gfCNCPoint2[10858] = {X 102.8887, Y 52.2397, Z -3.0000, A 0.000, B 0.000, C 0.000 }
gfCNCPoint2[10859] = {X 101.6641, Y 52.2655, Z -3.0000, A 0.000, B 0.000, C 0.000 }
gfCNCPoint2[10860] = {X 100.4526, Y 52.0855, Z -3.0000, A 0.000, B 0.000, C 0.000 }
gfCNCPoint2[10861] = {X 99.2883, Y 51.7050, Z -3.0000, A 0.000, B 0.000, C 0.000 }
gfCNCPoint2[10862] = {X 98.2043, Y 51.1347, Z -3.0000, A 0.000, B 0.000, C 0.000 }
gfCNCPoint2[10863] = {X 97.2313, Y 50.3907, Z -3.0000, A 0.000, B 0.000, C 0.000 }
gfCNCPoint2[10864] = {X 96.3865, Y 51.0508, Z -3.0000, A 0.000, B 0.000, C 0.000 }
gfCNCPoint2[10865] = {X 95.4539, Y 51.5797, Z -3.0000, A 0.000, B 0.000, C 0.000 }
gfCNCPoint2[10866] = {X 94.4538, Y 51.9659, Z -3.0000, A 0.000, B 0.000, C 0.000 }
gfCNCPoint2[10867] = {X 93.4078, Y 52.2011, Z -3.0000, A 0.000, B 0.000, C 0.000 }
gfCNCPoint2[10868] = {X 92.3385, Y 52.2800, Z -3.0000, A 0.000, B 0.000, C 0.000 }
gfCNCPoint2[10869] = {X 85.8951, Y 52.2800, Z -3.0000, A 0.000, B 0.000, C 0.000 }
gfCNCPoint2[10870] = {X 84.6852, Y 52.1788, Z -3.0000, A 0.000, B 0.000, C 0.000 }
gfCNCPoint2[10871] = {X 83.5090, Y 51.8779, Z -3.0000, A 0.000, B 0.000, C 0.000 }
gfCNCPoint2[10872] = {X 82.3992, Y 51.3857, Z -3.0000, A 0.000, B 0.000, C 0.000 }
gfCNCPoint2[10873] = {X 81.3866, Y 50.7159, Z -3.0000, A 0.000, B 0.000, C 0.000 }
gfCNCPoint2[10874] = {X 80.5223, Y 52.0937, Z -3.0000, A 0.000, B 0.000, C 0.000 }
gfCNCPoint2[10875] = {X 79.4808, Y 53.3429, Z -3.0000, A 0.000, B 0.000, C 0.000 }
gfCNCPoint2[10876] = {X 78.2809, Y 54.4408, Z -3.0000, A 0.000, B 0.000, C 0.000 }
gfCNCPoint2[10877] = {X 76.9444, Y 55.3676, Z -3.0000, A 0.000, B 0.000, C 0.000 }
gfCNCPoint2[10878] = {X 75.4955, Y 56.1065, Z -3.0000, A 0.000, B 0.000, C 0.000 }
gfCNCPoint2[10879] = {X 73.9605, Y 56.6440, Z -3.0000, A 0.000, B 0.000, C 0.000 }
gfCNCPoint2[10880] = {X 72.3672, Y 56.9705, Z -3.0000, A 0.000, B 0.000, C 0.000 }
gfCNCPoint2[10881] = {X 70.7445, Y 57.0800, Z -3.0000, A 0.000, B 0.000, C 0.000 }
gfCNCPoint2[10882] = {X 64.1851, Y 57.0800, Z -3.0000, A 0.000, B 0.000, C 0.000 }
gfCNCPoint2[10883] = {X 62.6628, Y 56.9837, Z -3.0000, A 0.000, B 0.000, C 0.000 }
gfCNCPoint2[10884] = {X 61.1646, Y 56.6963, Z -3.0000, A 0.000, B 0.000, C 0.000 }
gfCNCPoint2[10885] = {X 59.7147, Y 56.2224, Z -3.0000, A 0.000, B 0.000, C 0.000 }
gfCNCPoint2[10886] = {X 58.3360, Y 55.5695, Z -3.0000, A 0.000, B 0.000, C 0.000 }
gfCNCPoint2[10887] = {X 57.0507, Y 54.7481, Z -3.0000, A 0.000, B 0.000, C 0.000 }
gfCNCPoint2[10888] = {X 55.8790, Y 53.7713, Z -3.0000, A 0.000, B 0.000, C 0.000 }
gfCNCPoint2[10889] = {X 54.7074, Y 54.7481, Z -3.0000, A 0.000, B 0.000, C 0.000 }
gfCNCPoint2[10890] = {X 53.4220, Y 55.5695, Z -3.0000, A 0.000, B 0.000, C 0.000 }
gfCNCPoint2[10891] = {X 52.0434, Y 56.2224, Z -3.0000, A 0.000, B 0.000, C 0.000 }
gfCNCPoint2[10892] = {X 50.5934, Y 56.6963, Z -3.0000, A 0.000, B 0.000, C 0.000 }
gfCNCPoint2[10893] = {X 49.0953, Y 56.9837, Z -3.0000, A 0.000, B 0.000, C 0.000 }
gfCNCPoint2[10894] = {X 47.5729, Y 57.0800, Z -3.0000, A 0.000, B 0.000, C 0.000 }
gfCNCPoint2[10895] = {X 40.6393, Y 57.0800, Z -3.0000, A 0.000, B 0.000, C 0.000 }
gfCNCPoint2[10896] = {X 39.3237, Y 57.0081, Z -3.0000, A 0.000, B 0.000, C 0.000 }
gfCNCPoint2[10897] = {X 38.0238, Y 56.7934, Z -3.0000, A 0.000, B 0.000, C 0.000 }
gfCNCPoint2[10898] = {X 36.7550, Y 56.4385, Z -3.0000, A 0.000, B 0.000, C 0.000 }
gfCNCPoint2[10899] = {X 35.5323, Y 55.9474, Z -3.0000, A 0.000, B 0.000, C 0.000 }
gfCNCPoint2[10900] = {X 34.1223, Y 56.7816, Z -3.0000, A 0.000, B 0.000, C 0.000 }
gfCNCPoint2[10901] = {X 32.6361, Y 57.4711, Z -3.0000, A 0.000, B 0.000, C 0.000 }
gfCNCPoint2[10902] = {X 31.0886, Y 58.0091, Z -3.0000, A 0.000, B 0.000, C 0.000 }
gfCNCPoint2[10903] = {X 29.4952, Y 58.3901, Z -3.0000, A 0.000, B 0.000, C 0.000 }
gfCNCPoint2[10904] = {X 27.8718, Y 58.6104, Z -3.0000, A 0.000, B 0.000, C 0.000 }
gfCNCPoint2[10905] = {X 26.1298, Y 59.3568, Z -3.0000, A 0.000, B 0.000, C 0.000 }
gfCNCPoint2[10906] = {X 24.3546, Y 60.0200, Z -3.0000, A 0.000, B 0.000, C 0.000 }
gfCNCPoint2[10907] = {X 21.9380, Y 60.7953, Z -3.0000, A 0.000, B 0.000, C 0.000 }
gfCNCPoint2[10908] = {X 19.4715, Y 61.3930, Z -3.0000, A 0.000, B 0.000, C 0.000 }
gfCNCPoint2[10909] = {X 16.9680, Y 61.8098, Z -3.0000, A 0.000, B 0.000, C 0.000 }
gfCNCPoint2[10910] = {X 14.4409, Y 62.0436, Z -3.0000, A 0.000, B 0.000, C 0.000 }
gfCNCPoint2[10911] = {X 11.9035, Y 62.0931, Z -3.0000, A 0.000, B 0.000, C 0.000 }
gfCNCPoint2[10912] = {X 11.9035, Y 88.0950, Z -3.0000, A 0.000, B 0.000, C 0.000 }
gfCNCPoint2[10913] = {X 113.6337, Y 88.0950, Z -3.0000, A 0.000, B 0.000, C 0.000 }
gfCNCPoint2[10914] = {X 114.7670, Y 86.8212, Z -3.0000, A 0.000, B 0.000, C 0.000 }
gfCNCPoint2[10915] = {X 116.0421, Y 85.6894, Z -3.0000, A 0.000, B 0.000, C 0.000 }
gfCNCPoint2[10916] = {X 117.4414, Y 84.7153, Z -3.0000, A 0.000, B 0.000, C 0.000 }
gfCNCPoint2[10917] = {X 118.9454, Y 83.9125, Z -3.0000, A 0.000, B 0.000, C 0.000 }
gfCNCPoint2[10918] = {X 120.5335, Y 83.2920, Z -3.0000, A 0.000, B 0.000, C 0.000 }
gfCNCPoint2[10919] = {X 122.1834, Y 82.8625, Z -3.0000, A 0.000, B 0.000, C 0.000 }
gfCNCPoint2[10920] = {X 144.8180, Y 58.0066, Z -3.0000, A 0.000, B 0.000, C 0.000 }
gfCNCPoint2[10921] = {X 144.9143, Y 56.3321, Z -3.0000, A 0.000, B 0.000, C 0.000 }
gfCNCPoint2[10922] = {X 145.2037, Y 54.6800, Z -3.0000, A 0.000, B 0.000, C 0.000 }
gfCNCPoint2[10923] = {X 143.0396, Y 54.6800, Z -3.0000, A 0.000, B 0.000, C 0.000 }
gfCNCPoint2[10924] = {X 142.7952, Y 54.6769, Z -3.0000, A 0.000, B 0.000, C 0.000 }
gfCNCPoint2[10925] = {X 142.5510, Y 54.6677, Z -3.0000, A 0.000, B 0.000, C 0.000 }
gfCNCPoint2[10926] = {X 141.0979, Y 54.4832, Z -3.0000, A 0.000, B 0.000, C 0.000 }
gfCNCPoint2[10927] = {X 139.6893, Y 54.0817, Z -3.0000, A 0.000, B 0.000, C 0.000 }
gfCNCPoint2[10928] = {X 138.3574, Y 53.4722, Z -3.0000, A 0.000, B 0.000, C 0.000 }
gfCNCPoint2[10929] = {X 137.1327, Y 52.6688, Z -3.0000, A 0.000, B 0.000, C 0.000 }
gfCNCPoint2[10930] = {X 136.0432, Y 51.6898, Z -3.0000, A 0.000, B 0.000, C 0.000 }
gfCNCPoint2[10931] = {X 135.1140, Y 50.5575, Z -3.0000, A 0.000, B 0.000, C 0.000 }
gfCNCPoint2[10932] = {X 134.3662, Y 49.2981, Z -3.0000, A 0.000, B 0.000, C 0.000 }
gfCNCPoint2[10933] = {X 133.8170, Y 47.9402, Z -3.0000, A 0.000, B 0.000, C 0.000 }
gfCNCPoint2[10934] = {X 133.4789, Y 46.5151, Z -3.0000, A 0.000, B 0.000, C 0.000 }
gfCNCPoint2[10935] = {X 133.3598, Y 45.0552, Z -3.0000, A 0.000, B 0.000, C 0.000 }
gfCNCPoint2[10936] = {X 133.3601, Y 44.1105, Z -3.0000, A 0.000, B 0.000, C 0.000 }
gfCNCPoint2[10937] = {X 133.4665, Y 42.7743, Z -3.0000, A 0.000, B 0.000, C 0.000 }
gfCNCPoint2[10938] = {X 133.7565, Y 41.4655, Z -3.0000, A 0.000, B 0.000, C 0.000 }
gfCNCPoint2[10939] = {X 136.0581, Y 42.1457, Z -3.0000, A 0.000, B 0.000, C 0.000 }
gfCNCPoint2[10940] = {X 136.3664, Y 41.2990, Z -3.0000, A 0.000, B 0.000, C 0.000 }
gfCNCPoint2[10941] = {X 136.7770, Y 40.4969, Z -3.0000, A 0.000, B 0.000, C 0.000 }
gfCNCPoint2[10942] = {X 137.2836, Y 39.7516, Z -3.0000, A 0.000, B 0.000, C 0.000 }
gfCNCPoint2[10943] = {X 137.2836, Y 23.8768, Z -3.0000, A 0.000, B 0.000, C 0.000 }
gfCNCPoint2[10944] = {X 136.4352, Y 24.2641, Z -3.0000, A 0.000, B 0.000, C 0.000 }
gfCNCPoint2[10945] = {X 135.5443, Y 24.5398, Z -3.0000, A 0.000, B 0.000, C 0.000 }
gfCNCPoint2[10946] = {X 134.6254, Y 24.6993, Z -3.0000, A 0.000, B 0.000, C 0.000 }
gfCNCPoint2[10947] = {X 134.2595, Y 24.7296, Z -3.0000, A 0.000, B 0.000, C 0.000 }
gfCNCPoint2[10948] = {X 133.8926, Y 24.7414, Z -3.0000, A 0.000, B 0.000, C 0.000 }
gfCNCPoint2[10949] = {X 133.2006, Y 24.7415, Z -3.0000, A 0.000, B 0.000, C 0.000 }
gfCNCPoint2[10950] = {X 131.9926, Y 24.6406, Z -3.0000, A 0.000, B 0.000, C 0.000 }
gfCNCPoint2[10951] = {X 130.8180, Y 24.3406, Z -3.0000, A 0.000, B 0.000, C 0.000 }
gfCNCPoint2[10952] = {X 129.7095, Y 23.8498, Z -3.0000, A 0.000, B 0.000, C 0.000 }
gfCNCPoint2[10953] = {X 128.6978, Y 23.1819, Z -3.0000, A 0.000, B 0.000, C 0.000 }
gfCNCPoint2[10954] = {X 127.8110, Y 22.3554, Z -3.0000, A 0.000, B 0.000, C 0.000 }
gfCNCPoint2[10955] = {X 127.0736, Y 21.3931, Z -3.0000, A 0.000, B 0.000, C 0.000 }
gfCNCPoint2[10956] = {X 126.5061, Y 20.3219, Z -3.0000, A 0.000, B 0.000, C 0.000 }
gfCNCPoint2[10957] = {X 126.1243, Y 19.1713, Z -3.0000, A 0.000, B 0.000, C 0.000 }
gfCNCPoint2[10958] = {X 125.9387, Y 17.9733, Z -3.0000, A 0.000, B 0.000, C 0.000 }
gfCNCPoint2[10959] = {X 125.9251, Y 17.7176, Z -3.0000, A 0.000, B 0.000, C 0.000 }
gfCNCPoint2[10960] = {X 125.9206, Y 17.4615, Z -3.0000, A 0.000, B 0.000, C 0.000 }
gfCNCPoint2[10961] = {X 125.9206, Y 10.4835, Z -3.0000, A 0.000, B 0.000, C 0.000 }
gfCNCPoint2[10962] = {X 125.9372, Y 9.9932, Z -3.0000, A 0.000, B 0.000, C 0.000 }
gfCNCPoint2[10963] = {X 125.9867, Y 9.5050, Z -3.0000, A 0.000, B 0.000, C 0.000 }
gfCNCPoint2[10964] = {X 121.8686, Y 9.5050, Z -3.0000, A 0.000, B 0.000, C 0.000 }
gfCNCPoint2[10965] = {X 122.3091, Y 10.3411, Z -3.0000, A 0.000, B 0.000, C 0.000 }
gfCNCPoint2[10966] = {X 122.5801, Y 11.2463, Z -3.0000, A 0.000, B 0.000, C 0.000 }
gfCNCPoint2[10967] = {X 122.6716, Y 12.1868, Z -3.0000, A 0.000, B 0.000, C 0.000 }
gfCNCPoint2[10968] = {X 122.6714, Y 13.0237, Z -3.0000, A 0.000, B 0.000, C 0.000 }
gfCNCPoint2[10969] = {X 122.5640, Y 13.9970, Z -3.0000, A 0.000, B 0.000, C 0.000 }
gfCNCPoint2[10970] = {X 122.2645, Y 14.9292, Z -3.0000, A 0.000, B 0.000, C 0.000 }
gfCNCPoint2[10971] = {X 121.7850, Y 15.7828, Z -3.0000, A 0.000, B 0.000, C 0.000 }
gfCNCPoint2[10972] = {X 121.1447, Y 16.5236, Z -3.0000, A 0.000, B 0.000, C 0.000 }
gfCNCPoint2[10973] = {X 121.1435, Y 40.6621, Z -3.0000, A 0.000, B 0.000, C 0.000 }
gfCNCPoint2[10974] = {X 121.7851, Y 41.4041, Z -3.0000, A 0.000, B 0.000, C 0.000 }
gfCNCPoint2[10975] = {X 122.2653, Y 42.2595, Z -3.0000, A 0.000, B 0.000, C 0.000 }
gfCNCPoint2[10976] = {X 122.5648, Y 43.1936, Z -3.0000, A 0.000, B 0.000, C 0.000 }
gfCNCPoint2[10977] = {X 122.6714, Y 44.1688, Z -3.0000, A 0.000, B 0.000, C 0.000 }
gfCNCPoint2[10978] = {X 122.6716, Y 45.0000, Z -3.0000, A 0.000, B 0.000, C 0.000 }
gfCNCPoint2[10979] = {X 122.5778, Y 45.9520, Z -3.0000, A 0.000, B 0.000, C 0.000 }
gfCNCPoint2[10980] = {X 122.3001, Y 46.8675, Z -3.0000, A 0.000, B 0.000, C 0.000 }
gfCNCPoint2[10981] = {X 121.8491, Y 47.7112, Z -3.0000, A 0.000, B 0.000, C 0.000 }
gfCNCPoint2[10982] = {X 121.2423, Y 48.4507, Z -3.0000, A 0.000, B 0.000, C 0.000 }
gfCNCPoint2[10983] = {X 120.5028, Y 49.0576, Z -3.0000, A 0.000, B 0.000, C 0.000 }
gfCNCPoint2[10984] = {X 119.6591, Y 49.5085, Z -3.0000, A 0.000, B 0.000, C 0.000 }
gfCNCPoint2[10985] = {X 118.7436, Y 49.7862, Z -3.0000, A 0.000, B 0.000, C 0.000 }
gfCNCPoint2[10986] = {X 117.7916, Y 49.8800, Z -3.0000, A 0.000, B 0.000, C 0.000 }
gfCNCPoint2[10987] = {X 111.9185, Y 49.8800, Z -3.0000, A 0.000, B 0.000, C 0.000 }
gfCNCPoint2[10988] = {X 111.0234, Y 49.7972, Z -3.0000, A 0.000, B 0.000, C 0.000 }
gfCNCPoint2[10989] = {X 110.1587, Y 49.5517, Z -3.0000, A 0.000, B 0.000, C 0.000 }
gfCNCPoint2[10990] = {X 109.3537, Y 49.1517, Z -3.0000, A 0.000, B 0.000, C 0.000 }
gfCNCPoint2[10991] = {X 108.6357, Y 48.6108, Z -3.0000, A 0.000, B 0.000, C 0.000 }
gfCNCPoint2[10992] = {X 108.0714, Y 48.0024, Z -3.0000, A 0.000, B 0.000, C 0.000 }
gfCNCPoint2[10993] = {X 107.6183, Y 47.3071, Z -3.0000, A 0.000, B 0.000, C 0.000 }
gfCNCPoint2[10994] = {X 107.2895, Y 46.5451, Z -3.0000, A 0.000, B 0.000, C 0.000 }
gfCNCPoint2[10995] = {X 107.0947, Y 45.7384, Z -3.0000, A 0.000, B 0.000, C 0.000 }
gfCNCPoint2[10996] = {X 106.6287, Y 46.8769, Z -3.0000, A 0.000, B 0.000, C 0.000 }
gfCNCPoint2[10997] = {X 106.1131, Y 47.8110, Z -3.0000, A 0.000, B 0.000, C 0.000 }
gfCNCPoint2[10998] = {X 105.4068, Y 48.6108, Z -3.0000, A 0.000, B 0.000, C 0.000 }
gfCNCPoint2[10999] = {X 104.8391, Y 49.0550, Z -3.0000, A 0.000, B 0.000, C 0.000 }
gfCNCPoint2[11000] = {X 104.2121, Y 49.4107, Z -3.0000, A 0.000, B 0.000, C 0.000 }
gfCNCPoint2[11001] = {X 103.3106, Y 49.7335, Z -3.0000, A 0.000, B 0.000, C 0.000 }
gfCNCPoint2[11002] = {X 102.3635, Y 49.8741, Z -3.0000, A 0.000, B 0.000, C 0.000 }
gfCNCPoint2[11003] = {X 101.4071, Y 49.8271, Z -3.0000, A 0.000, B 0.000, C 0.000 }
gfCNCPoint2[11004] = {X 100.4784, Y 49.5941, Z -3.0000, A 0.000, B 0.000, C 0.000 }
gfCNCPoint2[11005] = {X 99.6130, Y 49.1844, Z -3.0000, A 0.000, B 0.000, C 0.000 }
gfCNCPoint2[11006] = {X 98.8443, Y 48.6135, Z -3.0000, A 0.000, B 0.000, C 0.000 }
gfCNCPoint2[11007] = {X 98.1362, Y 47.8127, Z -3.0000, A 0.000, B 0.000, C 0.000 }
gfCNCPoint2[11008] = {X 97.6194, Y 46.8769, Z -3.0000, A 0.000, B 0.000, C 0.000 }
gfCNCPoint2[11009] = {X 97.1600, Y 45.7536, Z -3.0000, A 0.000, B 0.000, C 0.000 }
gfCNCPoint2[11010] = {X 96.9635, Y 46.5570, Z -3.0000, A 0.000, B 0.000, C 0.000 }
gfCNCPoint2[11011] = {X 96.6342, Y 47.3156, Z -3.0000, A 0.000, B 0.000, C 0.000 }
gfCNCPoint2[11012] = {X 96.1814, Y 48.0078, Z -3.0000, A 0.000, B 0.000, C 0.000 }
gfCNCPoint2[11013] = {X 95.6183, Y 48.6135, Z -3.0000, A 0.000, B 0.000, C 0.000 }
gfCNCPoint2[11014] = {X 94.9007, Y 49.1533, Z -3.0000, A 0.000, B 0.000, C 0.000 }
gfCNCPoint2[11015] = {X 94.0964, Y 49.5524, Z -3.0000, A 0.000, B 0.000, C 0.000 }
gfCNCPoint2[11016] = {X 93.2326, Y 49.7974, Z -3.0000, A 0.000, B 0.000, C 0.000 }
gfCNCPoint2[11017] = {X 92.3385, Y 49.8800, Z -3.0000, A 0.000, B 0.000, C 0.000 }
gfCNCPoint2[11018] = {X 85.8951, Y 49.8800, Z -3.0000, A 0.000, B 0.000, C 0.000 }
gfCNCPoint2[11019] = {X 85.0841, Y 49.8121, Z -3.0000, A 0.000, B 0.000, C 0.000 }
gfCNCPoint2[11020] = {X 84.2956, Y 49.6104, Z -3.0000, A 0.000, B 0.000, C 0.000 }
gfCNCPoint2[11021] = {X 83.5517, Y 49.2805, Z -3.0000, A 0.000, B 0.000, C 0.000 }
gfCNCPoint2[11022] = {X 82.8729, Y 48.8316, Z -3.0000, A 0.000, B 0.000, C 0.000 }
gfCNCPoint2[11023] = {X 82.2391, Y 48.2324, Z -3.0000, A 0.000, B 0.000, C 0.000 }
gfCNCPoint2[11024] = {X 81.7221, Y 47.5300, Z -3.0000, A 0.000, B 0.000, C 0.000 }
gfCNCPoint2[11025] = {X 81.3384, Y 46.7467, Z -3.0000, A 0.000, B 0.000, C 0.000 }
gfCNCPoint2[11026] = {X 81.1002, Y 45.9077, Z -3.0000, A 0.000, B 0.000, C 0.000 }
gfCNCPoint2[11027] = {X 81.0152, Y 45.0397, Z -3.0000, A 0.000, B 0.000, C 0.000 }
gfCNCPoint2[11028] = {X 81.0151, Y 44.2034, Z -3.0000, A 0.000, B 0.000, C 0.000 }
gfCNCPoint2[11029] = {X 81.1203, Y 43.2199, Z -3.0000, A 0.000, B 0.000, C 0.000 }
gfCNCPoint2[11030] = {X 81.4192, Y 42.2770, Z -3.0000, A 0.000, B 0.000, C 0.000 }
gfCNCPoint2[11031] = {X 81.9000, Y 41.4125, Z -3.0000, A 0.000, B 0.000, C 0.000 }
gfCNCPoint2[11032] = {X 82.5434, Y 40.6612, Z -3.0000, A 0.000, B 0.000, C 0.000 }
gfCNCPoint2[11033] = {X 82.5432, Y 25.2537, Z -3.0000, A 0.000, B 0.000, C 0.000 }
gfCNCPoint2[11034] = {X 77.7432, Y 25.2537, Z -3.0000, A 0.000, B 0.000, C 0.000 }
gfCNCPoint2[11035] = {X 77.7431, Y 18.1980, Z -3.0000, A 0.000, B 0.000, C 0.000 }
gfCNCPoint2[11036] = {X 77.0784, Y 16.9741, Z -3.0000, A 0.000, B 0.000, C 0.000 }
gfCNCPoint2[11037] = {X 76.5962, Y 15.6674, Z -3.0000, A 0.000, B 0.000, C 0.000 }
gfCNCPoint2[11038] = {X 76.3065, Y 14.3050, Z -3.0000, A 0.000, B 0.000, C 0.000 }
gfCNCPoint2[11039] = {X 74.0412, Y 14.3050, Z -3.0000, A 0.000, B 0.000, C 0.000 }
gfCNCPoint2[11040] = {X 73.9992, Y 14.7015, Z -3.0000, A 0.000, B 0.000, C 0.000 }
gfCNCPoint2[11041] = {X 73.9463, Y 15.0967, Z -3.0000, A 0.000, B 0.000, C 0.000 }
gfCNCPoint2[11042] = {X 77.7432, Y 25.2537, Z -3.0000, A 0.000, B 0.000, C 0.000 }
gfCNCPoint2[11043] = {X 80.1432, Y 25.2537, Z -3.0000, A 0.000, B 0.000, C 0.000 }
gfCNCPoint2[11044] = {X 80.1431, Y 17.4405, Z -3.0000, A 0.000, B 0.000, C 0.000 }
gfCNCPoint2[11045] = {X 79.4946, Y 16.4468, Z -3.0000, A 0.000, B 0.000, C 0.000 }
gfCNCPoint2[11046] = {X 79.0161, Y 15.3611, Z -3.0000, A 0.000, B 0.000, C 0.000 }
gfCNCPoint2[11047] = {X 78.7204, Y 14.2120, Z -3.0000, A 0.000, B 0.000, C 0.000 }
gfCNCPoint2[11048] = {X 78.6153, Y 13.0301, Z -3.0000, A 0.000, B 0.000, C 0.000 }
gfCNCPoint2[11049] = {X 78.6151, Y 12.1868, Z -3.0000, A 0.000, B 0.000, C 0.000 }
gfCNCPoint2[11050] = {X 78.6164, Y 12.0459, Z -3.0000, A 0.000, B 0.000, C 0.000 }
gfCNCPoint2[11051] = {X 78.6205, Y 11.9050, Z -3.0000, A 0.000, B 0.000, C 0.000 }
gfCNCPoint2[11052] = {X 71.6988, Y 11.9050, Z -3.0000, A 0.000, B 0.000, C 0.000 }
gfCNCPoint2[11053] = {X 71.7013, Y 12.0459, Z -3.0000, A 0.000, B 0.000, C 0.000 }
gfCNCPoint2[11054] = {X 71.7021, Y 12.1868, Z -3.0000, A 0.000, B 0.000, C 0.000 }
gfCNCPoint2[11055] = {X 71.7016, Y 13.0911, Z -3.0000, A 0.000, B 0.000, C 0.000 }
gfCNCPoint2[11056] = {X 71.6385, Y 14.2157, Z -3.0000, A 0.000, B 0.000, C 0.000 }
gfCNCPoint2[11057] = {X 71.4711, Y 15.3294, Z -3.0000, A 0.000, B 0.000, C 0.000 }
gfCNCPoint2[11058] = {X 78.9542, Y 35.3473, Z -3.0000, A 0.000, B 0.000, C 0.000 }
gfCNCPoint2[11059] = {X 79.5718, Y 35.9623, Z -3.0000, A 0.000, B 0.000, C 0.000 }
gfCNCPoint2[11060] = {X 80.1433, Y 36.6202, Z -3.0000, A 0.000, B 0.000, C 0.000 }
gfCNCPoint2[11061] = {X 80.1432, Y 25.2537, Z -3.0000, A 0.000, B 0.000, C 0.000 }
gfCNCPoint2[11062] = {X 82.5432, Y 25.2537, Z -3.0000, A 0.000, B 0.000, C 0.000 }
gfCNCPoint2[11063] = {X 82.5431, Y 16.5247, Z -3.0000, A 0.000, B 0.000, C 0.000 }
gfCNCPoint2[11064] = {X 81.9017, Y 15.7830, Z -3.0000, A 0.000, B 0.000, C 0.000 }
gfCNCPoint2[11065] = {X 81.4216, Y 14.9280, Z -3.0000, A 0.000, B 0.000, C 0.000 }
gfCNCPoint2[11066] = {X 81.1221, Y 13.9943, Z -3.0000, A 0.000, B 0.000, C 0.000 }
gfCNCPoint2[11067] = {X 81.0153, Y 13.0196, Z -3.0000, A 0.000, B 0.000, C 0.000 }
gfCNCPoint2[11068] = {X 81.0151, Y 12.1868, Z -3.0000, A 0.000, B 0.000, C 0.000 }
gfCNCPoint2[11069] = {X 81.0160, Y 12.0924, Z -3.0000, A 0.000, B 0.000, C 0.000 }
gfCNCPoint2[11070] = {X 81.0187, Y 11.9979, Z -3.0000, A 0.000, B 0.000, C 0.000 }
gfCNCPoint2[11071] = {X 81.1324, Y 11.1230, Z -3.0000, A 0.000, B 0.000, C 0.000 }
gfCNCPoint2[11072] = {X 81.4018, Y 10.2829, Z -3.0000, A 0.000, B 0.000, C 0.000 }
gfCNCPoint2[11073] = {X 81.8180, Y 9.5050, Z -3.0000, A 0.000, B 0.000, C 0.000 }
gfCNCPoint2[11074] = {X 82.2190, Y 9.7688, Z -3.0000, A 0.000, B 0.000, C 0.000 }
gfCNCPoint2[11075] = {X 82.7659, Y 9.0936, Z -3.0000, A 0.000, B 0.000, C 0.000 }
gfCNCPoint2[11076] = {X 83.4347, Y 8.5390, Z -3.0000, A 0.000, B 0.000, C 0.000 }
gfCNCPoint2[11077] = {X 84.1995, Y 8.1266, Z -3.0000, A 0.000, B 0.000, C 0.000 }
gfCNCPoint2[11078] = {X 85.0304, Y 7.8726, Z -3.0000, A 0.000, B 0.000, C 0.000 }
gfCNCPoint2[11079] = {X 85.8951, Y 7.7868, Z -3.0000, A 0.000, B 0.000, C 0.000 }
gfCNCPoint2[11080] = {X 94.0497, Y 7.7868, Z -3.0000, A 0.000, B 0.000, C 0.000 }
gfCNCPoint2[11081] = {X 95.0288, Y 7.8971, Z -3.0000, A 0.000, B 0.000, C 0.000 }
gfCNCPoint2[11082] = {X 95.9588, Y 8.2226, Z -3.0000, A 0.000, B 0.000, C 0.000 }
gfCNCPoint2[11083] = {X 96.7930, Y 8.7468, Z -3.0000, A 0.000, B 0.000, C 0.000 }
gfCNCPoint2[11084] = {X 97.4897, Y 9.4435, Z -3.0000, A 0.000, B 0.000, C 0.000 }
gfCNCPoint2[11085] = {X 98.0139, Y 10.2777, Z -3.0000, A 0.000, B 0.000, C 0.000 }
gfCNCPoint2[11086] = {X 98.3394, Y 11.2077, Z -3.0000, A 0.000, B 0.000, C 0.000 }
gfCNCPoint2[11087] = {X 98.4497, Y 12.1868, Z -3.0000, A 0.000, B 0.000, C 0.000 }
gfCNCPoint2[11088] = {X 98.4494, Y 13.0233, Z -3.0000, A 0.000, B 0.000, C 0.000 }
gfCNCPoint2[11089] = {X 98.3723, Y 13.7994, Z -3.0000, A 0.000, B 0.000, C 0.000 }
gfCNCPoint2[11090] = {X 98.1594, Y 14.5497, Z -3.0000, A 0.000, B 0.000, C 0.000 }
gfCNCPoint2[11091] = {X 97.8174, Y 15.2505, Z -3.0000, A 0.000, B 0.000, C 0.000 }
gfCNCPoint2[11092] = {X 98.3672, Y 16.6193, Z -3.0000, A 0.000, B 0.000, C 0.000 }
gfCNCPoint2[11093] = {X 101.8765, Y 25.3184, Z -3.0000, A 0.000, B 0.000, C 0.000 }
gfCNCPoint2[11094] = {X 105.9244, Y 15.2235, Z -3.0000, A 0.000, B 0.000, C 0.000 }
gfCNCPoint2[11095] = {X 105.5858, Y 14.5158, Z -3.0000, A 0.000, B 0.000, C 0.000 }
gfCNCPoint2[11096] = {X 105.3782, Y 13.7593, Z -3.0000, A 0.000, B 0.000, C 0.000 }
gfCNCPoint2[11097] = {X 105.3083, Y 12.9779, Z -3.0000, A 0.000, B 0.000, C 0.000 }
gfCNCPoint2[11098] = {X 105.3083, Y 12.1868, Z -3.0000, A 0.000, B 0.000, C 0.000 }
gfCNCPoint2[11099] = {X 105.4186, Y 11.2077, Z -3.0000, A 0.000, B 0.000, C 0.000 }
gfCNCPoint2[11100] = {X 105.7440, Y 10.2777, Z -3.0000, A 0.000, B 0.000, C 0.000 }
gfCNCPoint2[11101] = {X 106.2682, Y 9.4435, Z -3.0000, A 0.000, B 0.000, C 0.000 }
gfCNCPoint2[11102] = {X 106.9649, Y 8.7468, Z -3.0000, A 0.000, B 0.000, C 0.000 }
gfCNCPoint2[11103] = {X 107.7992, Y 8.2226, Z -3.0000, A 0.000, B 0.000, C 0.000 }
gfCNCPoint2[11104] = {X 108.7292, Y 7.8971, Z -3.0000, A 0.000, B 0.000, C 0.000 }
gfCNCPoint2[11105] = {X 109.7083, Y 7.7868, Z -3.0000, A 0.000, B 0.000, C 0.000 }
gfCNCPoint2[11106] = {X 117.7916, Y 7.7868, Z -3.0000, A 0.000, B 0.000, C 0.000 }
gfCNCPoint2[11107] = {X 118.7707, Y 7.8971, Z -3.0000, A 0.000, B 0.000, C 0.000 }
gfCNCPoint2[11108] = {X 119.7007, Y 8.2226, Z -3.0000, A 0.000, B 0.000, C 0.000 }
gfCNCPoint2[11109] = {X 120.5349, Y 8.7468, Z -3.0000, A 0.000, B 0.000, C 0.000 }
gfCNCPoint2[11110] = {X 121.2316, Y 9.4435, Z -3.0000, A 0.000, B 0.000, C 0.000 }
gfCNCPoint2[11111] = {X 121.7558, Y 10.2777, Z -3.0000, A 0.000, B 0.000, C 0.000 }
gfCNCPoint2[11112] = {X 122.0813, Y 11.2077, Z -3.0000, A 0.000, B 0.000, C 0.000 }
gfCNCPoint2[11113] = {X 122.1916, Y 12.1868, Z -3.0000, A 0.000, B 0.000, C 0.000 }
gfCNCPoint2[11114] = {X 122.1913, Y 13.0233, Z -3.0000, A 0.000, B 0.000, C 0.000 }
gfCNCPoint2[11115] = {X 122.0831, Y 13.9491, Z -3.0000, A 0.000, B 0.000, C 0.000 }
gfCNCPoint2[11116] = {X 121.7822, Y 14.8314, Z -3.0000, A 0.000, B 0.000, C 0.000 }
gfCNCPoint2[11117] = {X 121.3022, Y 15.6305, Z -3.0000, A 0.000, B 0.000, C 0.000 }
gfCNCPoint2[11118] = {X 120.6647, Y 16.3105, Z -3.0000, A 0.000, B 0.000, C 0.000 }
gfCNCPoint2[11119] = {X 120.6635, Y 40.8758, Z -3.0000, A 0.000, B 0.000, C 0.000 }
gfCNCPoint2[11120] = {X 120.6784, Y 40.8882, Z -3.0000, A 0.000, B 0.000, C 0.000 }
gfCNCPoint2[11121] = {X 121.3172, Y 41.5763, Z -3.0000, A 0.000, B 0.000, C 0.000 }
gfCNCPoint2[11122] = {X 121.7955, Y 42.3843, Z -3.0000, A 0.000, B 0.000, C 0.000 }
gfCNCPoint2[11123] = {X 122.0914, Y 43.2754, Z -3.0000, A 0.000, B 0.000, C 0.000 }
gfCNCPoint2[11124] = {X 122.1916, Y 44.2089, Z -3.0000, A 0.000, B 0.000, C 0.000 }
gfCNCPoint2[11125] = {X 122.1916, Y 45.0000, Z -3.0000, A 0.000, B 0.000, C 0.000 }
gfCNCPoint2[11126] = {X 122.0813, Y 45.9791, Z -3.0000, A 0.000, B 0.000, C 0.000 }
gfCNCPoint2[11127] = {X 121.7558, Y 46.9091, Z -3.0000, A 0.000, B 0.000, C 0.000 }
gfCNCPoint2[11128] = {X 121.2316, Y 47.7434, Z -3.0000, A 0.000, B 0.000, C 0.000 }
gfCNCPoint2[11129] = {X 120.5349, Y 48.4401, Z -3.0000, A 0.000, B 0.000, C 0.000 }
gfCNCPoint2[11130] = {X 119.7007, Y 48.9643, Z -3.0000, A 0.000, B 0.000, C 0.000 }
gfCNCPoint2[11131] = {X 118.7707, Y 49.2897, Z -3.0000, A 0.000, B 0.000, C 0.000 }
gfCNCPoint2[11132] = {X 117.7916, Y 49.4000, Z -3.0000, A 0.000, B 0.000, C 0.000 }
gfCNCPoint2[11133] = {X 111.9185, Y 49.4000, Z -3.0000, A 0.000, B 0.000, C 0.000 }
gfCNCPoint2[11134] = {X 110.9394, Y 49.2897, Z -3.0000, A 0.000, B 0.000, C 0.000 }
gfCNCPoint2[11135] = {X 110.0094, Y 48.9643, Z -3.0000, A 0.000, B 0.000, C 0.000 }
gfCNCPoint2[11136] = {X 109.1751, Y 48.4400, Z -3.0000, A 0.000, B 0.000, C 0.000 }
gfCNCPoint2[11137] = {X 108.4784, Y 47.7433, Z -3.0000, A 0.000, B 0.000, C 0.000 }
gfCNCPoint2[11138] = {X 107.9542, Y 46.9091, Z -3.0000, A 0.000, B 0.000, C 0.000 }
gfCNCPoint2[11139] = {X 107.6288, Y 45.9791, Z -3.0000, A 0.000, B 0.000, C 0.000 }
gfCNCPoint2[11140] = {X 107.5185, Y 45.0000, Z -3.0000, A 0.000, B 0.000, C 0.000 }
gfCNCPoint2[11141] = {X 107.5185, Y 44.1811, Z -3.0000, A 0.000, B 0.000, C 0.000 }
gfCNCPoint2[11142] = {X 107.5551, Y 43.6251, Z -3.0000, A 0.000, B 0.000, C 0.000 }
gfCNCPoint2[11143] = {X 107.6644, Y 43.0786, Z -3.0000, A 0.000, B 0.000, C 0.000 }
gfCNCPoint2[11144] = {X 106.1856, Y 46.6923, Z -3.0000, A 0.000, B 0.000, C 0.000 }
gfCNCPoint2[11145] = {X 105.8087, Y 47.4049, Z -3.0000, A 0.000, B 0.000, C 0.000 }
gfCNCPoint2[11146] = {X 105.3081, Y 48.0367, Z -3.0000, A 0.000, B 0.000, C 0.000 }
gfCNCPoint2[11147] = {X 104.7006, Y 48.5667, Z -3.0000, A 0.000, B 0.000, C 0.000 }
gfCNCPoint2[11148] = {X 104.0067, Y 48.9769, Z -3.0000, A 0.000, B 0.000, C 0.000 }
gfCNCPoint2[11149] = {X 103.0414, Y 49.3033, Z -3.0000, A 0.000, B 0.000, C 0.000 }
gfCNCPoint2[11150] = {X 102.0269, Y 49.3989, Z -3.0000, A 0.000, B 0.000, C 0.000 }
gfCNCPoint2[11151] = {X 101.0176, Y 49.2586, Z -3.0000, A 0.000, B 0.000, C 0.000 }
gfCNCPoint2[11152] = {X 100.0676, Y 48.8899, Z -3.0000, A 0.000, B 0.000, C 0.000 }
gfCNCPoint2[11153] = {X 99.2280, Y 48.3125, Z -3.0000, A 0.000, B 0.000, C 0.000 }
gfCNCPoint2[11154] = {X 98.5436, Y 47.5575, Z -3.0000, A 0.000, B 0.000, C 0.000 }
gfCNCPoint2[11155] = {X 98.0514, Y 46.6653, Z -3.0000, A 0.000, B 0.000, C 0.000 }
gfCNCPoint2[11156] = {X 96.5861, Y 43.0817, Z -3.0000, A 0.000, B 0.000, C 0.000 }
gfCNCPoint2[11157] = {X 96.6982, Y 43.6405, Z -3.0000, A 0.000, B 0.000, C 0.000 }
gfCNCPoint2[11158] = {X 96.7385, Y 44.2089, Z -3.0000, A 0.000, B 0.000, C 0.000 }
gfCNCPoint2[11159] = {X 96.7383, Y 45.0423, Z -3.0000, A 0.000, B 0.000, C 0.000 }
gfCNCPoint2[11160] = {X 96.6200, Y 46.0144, Z -3.0000, A 0.000, B 0.000, C 0.000 }
gfCNCPoint2[11161] = {X 96.2896, Y 46.9363, Z -3.0000, A 0.000, B 0.000, C 0.000 }
gfCNCPoint2[11162] = {X 95.7635, Y 47.7622, Z -3.0000, A 0.000, B 0.000, C 0.000 }
gfCNCPoint2[11163] = {X 95.0677, Y 48.4513, Z -3.0000, A 0.000, B 0.000, C 0.000 }
gfCNCPoint2[11164] = {X 94.2367, Y 48.9695, Z -3.0000, A 0.000, B 0.000, C 0.000 }
gfCNCPoint2[11165] = {X 93.3117, Y 49.2910, Z -3.0000, A 0.000, B 0.000, C 0.000 }
gfCNCPoint2[11166] = {X 92.3385, Y 49.4000, Z -3.0000, A 0.000, B 0.000, C 0.000 }
gfCNCPoint2[11167] = {X 85.8951, Y 49.4000, Z -3.0000, A 0.000, B 0.000, C 0.000 }
gfCNCPoint2[11168] = {X 84.9160, Y 49.2897, Z -3.0000, A 0.000, B 0.000, C 0.000 }
gfCNCPoint2[11169] = {X 83.9860, Y 48.9643, Z -3.0000, A 0.000, B 0.000, C 0.000 }
gfCNCPoint2[11170] = {X 83.1517, Y 48.4400, Z -3.0000, A 0.000, B 0.000, C 0.000 }
gfCNCPoint2[11171] = {X 82.4550, Y 47.7433, Z -3.0000, A 0.000, B 0.000, C 0.000 }
gfCNCPoint2[11172] = {X 81.9308, Y 46.9091, Z -3.0000, A 0.000, B 0.000, C 0.000 }
gfCNCPoint2[11173] = {X 81.6054, Y 45.9791, Z -3.0000, A 0.000, B 0.000, C 0.000 }
gfCNCPoint2[11174] = {X 81.4951, Y 45.0000, Z -3.0000, A 0.000, B 0.000, C 0.000 }
gfCNCPoint2[11175] = {X 81.4951, Y 44.2064, Z -3.0000, A 0.000, B 0.000, C 0.000 }
gfCNCPoint2[11176] = {X 81.6006, Y 43.2693, Z -3.0000, A 0.000, B 0.000, C 0.000 }
gfCNCPoint2[11177] = {X 81.9008, Y 42.3753, Z -3.0000, A 0.000, B 0.000, C 0.000 }
gfCNCPoint2[11178] = {X 82.3823, Y 41.5644, Z -3.0000, A 0.000, B 0.000, C 0.000 }
gfCNCPoint2[11179] = {X 83.0234, Y 40.8728, Z -3.0000, A 0.000, B 0.000, C 0.000 }
gfCNCPoint2[11180] = {X 83.0231, Y 16.3115, Z -3.0000, A 0.000, B 0.000, C 0.000 }
gfCNCPoint2[11181] = {X 82.3783, Y 15.6223, Z -3.0000, A 0.000, B 0.000, C 0.000 }
gfCNCPoint2[11182] = {X 81.8953, Y 14.8115, Z -3.0000, A 0.000, B 0.000, C 0.000 }
gfCNCPoint2[11183] = {X 81.5963, Y 13.9163, Z -3.0000, A 0.000, B 0.000, C 0.000 }
gfCNCPoint2[11184] = {X 81.4951, Y 12.9779, Z -3.0000, A 0.000, B 0.000, C 0.000 }
gfCNCPoint2[11185] = {X 81.4951, Y 12.1868, Z -3.0000, A 0.000, B 0.000, C 0.000 }
gfCNCPoint2[11186] = {X 81.5776, Y 11.3388, Z -3.0000, A 0.000, B 0.000, C 0.000 }
gfCNCPoint2[11187] = {X 81.8219, Y 10.5226, Z -3.0000, A 0.000, B 0.000, C 0.000 }
gfCNCPoint2[11188] = {X 82.2190, Y 9.7688, Z -3.0000, A 0.000, B 0.000, C 0.000 }
gfCNCPoint2[11189] = {X 81.8180, Y 9.5050, Z -3.0000, A 0.000, B 0.000, C 0.000 }
gfCNCPoint2[11190] = {X 68.9232, Y 9.5050, Z -3.0000, A 0.000, B 0.000, C 0.000 }
gfCNCPoint2[11191] = {X 69.1905, Y 10.7209, Z -3.0000, A 0.000, B 0.000, C 0.000 }
gfCNCPoint2[11192] = {X 69.2995, Y 11.9610, Z -3.0000, A 0.000, B 0.000, C 0.000 }
gfCNCPoint2[11193] = {X 69.3015, Y 12.0739, Z -3.0000, A 0.000, B 0.000, C 0.000 }
gfCNCPoint2[11194] = {X 69.3021, Y 12.1868, Z -3.0000, A 0.000, B 0.000, C 0.000 }
gfCNCPoint2[11195] = {X 69.3017, Y 13.0686, Z -3.0000, A 0.000, B 0.000, C 0.000 }
gfCNCPoint2[11196] = {X 69.2126, Y 14.2911, Z -3.0000, A 0.000, B 0.000, C 0.000 }
gfCNCPoint2[11197] = {X 68.9698, Y 15.4926, Z -3.0000, A 0.000, B 0.000, C 0.000 }
gfCNCPoint2[11198] = {X 76.9173, Y 36.7523, Z -3.0000, A 0.000, B 0.000, C 0.000 }
gfCNCPoint2[11199] = {X 77.6311, Y 37.4061, Z -3.0000, A 0.000, B 0.000, C 0.000 }
gfCNCPoint2[11200] = {X 78.2760, Y 38.1278, Z -3.0000, A 0.000, B 0.000, C 0.000 }
gfCNCPoint2[11201] = {X 79.0234, Y 39.1926, Z -3.0000, A 0.000, B 0.000, C 0.000 }
gfCNCPoint2[11202] = {X 79.6212, Y 40.3480, Z -3.0000, A 0.000, B 0.000, C 0.000 }
gfCNCPoint2[11203] = {X 80.0587, Y 41.5731, Z -3.0000, A 0.000, B 0.000, C 0.000 }
gfCNCPoint2[11204] = {X 80.3280, Y 42.8459, Z -3.0000, A 0.000, B 0.000, C 0.000 }
gfCNCPoint2[11205] = {X 80.4242, Y 44.1432, Z -3.0000, A 0.000, B 0.000, C 0.000 }
gfCNCPoint2[11206] = {X 80.4245, Y 45.0000, Z -3.0000, A 0.000, B 0.000, C 0.000 }
gfCNCPoint2[11207] = {X 80.3511, Y 46.1898, Z -3.0000, A 0.000, B 0.000, C 0.000 }
gfCNCPoint2[11208] = {X 80.1320, Y 47.3615, Z -3.0000, A 0.000, B 0.000, C 0.000 }
gfCNCPoint2[11209] = {X 79.7706, Y 48.4974, Z -3.0000, A 0.000, B 0.000, C 0.000 }
gfCNCPoint2[11210] = {X 79.2722, Y 49.5803, Z -3.0000, A 0.000, B 0.000, C 0.000 }
gfCNCPoint2[11211] = {X 78.4688, Y 50.8341, Z -3.0000, A 0.000, B 0.000, C 0.000 }
gfCNCPoint2[11212] = {X 77.4826, Y 51.9498, Z -3.0000, A 0.000, B 0.000, C 0.000 }
gfCNCPoint2[11213] = {X 76.3369, Y 52.9011, Z -3.0000, A 0.000, B 0.000, C 0.000 }
gfCNCPoint2[11214] = {X 75.0589, Y 53.6653, Z -3.0000, A 0.000, B 0.000, C 0.000 }
gfCNCPoint2[11215] = {X 73.6787, Y 54.2246, Z -3.0000, A 0.000, B 0.000, C 0.000 }
gfCNCPoint2[11216] = {X 72.2292, Y 54.5655, Z -3.0000, A 0.000, B 0.000, C 0.000 }
gfCNCPoint2[11217] = {X 70.7445, Y 54.6800, Z -3.0000, A 0.000, B 0.000, C 0.000 }
gfCNCPoint2[11218] = {X 64.1851, Y 54.6800, Z -3.0000, A 0.000, B 0.000, C 0.000 }
gfCNCPoint2[11219] = {X 62.7229, Y 54.5689, Z -3.0000, A 0.000, B 0.000, C 0.000 }
gfCNCPoint2[11220] = {X 61.2943, Y 54.2383, Z -3.0000, A 0.000, B 0.000, C 0.000 }
gfCNCPoint2[11221] = {X 59.9320, Y 53.6956, Z -3.0000, A 0.000, B 0.000, C 0.000 }
gfCNCPoint2[11222] = {X 58.6673, Y 52.9534, Z -3.0000, A 0.000, B 0.000, C 0.000 }
gfCNCPoint2[11223] = {X 57.5293, Y 52.0286, Z -3.0000, A 0.000, B 0.000, C 0.000 }
gfCNCPoint2[11224] = {X 56.6337, Y 51.0563, Z -3.0000, A 0.000, B 0.000, C 0.000 }
gfCNCPoint2[11225] = {X 55.8790, Y 49.9710, Z -3.0000, A 0.000, B 0.000, C 0.000 }
gfCNCPoint2[11226] = {X 55.1243, Y 51.0563, Z -3.0000, A 0.000, B 0.000, C 0.000 }
gfCNCPoint2[11227] = {X 54.2288, Y 52.0286, Z -3.0000, A 0.000, B 0.000, C 0.000 }
gfCNCPoint2[11228] = {X 53.0907, Y 52.9534, Z -3.0000, A 0.000, B 0.000, C 0.000 }
gfCNCPoint2[11229] = {X 51.8261, Y 53.6956, Z -3.0000, A 0.000, B 0.000, C 0.000 }
gfCNCPoint2[11230] = {X 50.4638, Y 54.2383, Z -3.0000, A 0.000, B 0.000, C 0.000 }
gfCNCPoint2[11231] = {X 49.0351, Y 54.5689, Z -3.0000, A 0.000, B 0.000, C 0.000 }
gfCNCPoint2[11232] = {X 47.5729, Y 54.6800, Z -3.0000, A 0.000, B 0.000, C 0.000 }
gfCNCPoint2[11233] = {X 40.6393, Y 54.6800, Z -3.0000, A 0.000, B 0.000, C 0.000 }
gfCNCPoint2[11234] = {X 39.2448, Y 54.5790, Z -3.0000, A 0.000, B 0.000, C 0.000 }
gfCNCPoint2[11235] = {X 37.8793, Y 54.2782, Z -3.0000, A 0.000, B 0.000, C 0.000 }
gfCNCPoint2[11236] = {X 36.5715, Y 53.7838, Z -3.0000, A 0.000, B 0.000, C 0.000 }
gfCNCPoint2[11237] = {X 35.3485, Y 53.1062, Z -3.0000, A 0.000, B 0.000, C 0.000 }
gfCNCPoint2[11238] = {X 33.9161, Y 54.1337, Z -3.0000, A 0.000, B 0.000, C 0.000 }
gfCNCPoint2[11239] = {X 32.3660, Y 54.9733, Z -3.0000, A 0.000, B 0.000, C 0.000 }
gfCNCPoint2[11240] = {X 30.7228, Y 55.6116, Z -3.0000, A 0.000, B 0.000, C 0.000 }
gfCNCPoint2[11241] = {X 29.0125, Y 56.0387, Z -3.0000, A 0.000, B 0.000, C 0.000 }
gfCNCPoint2[11242] = {X 27.2621, Y 56.2477, Z -3.0000, A 0.000, B 0.000, C 0.000 }
gfCNCPoint2[11243] = {X 25.4278, Y 57.0520, Z -3.0000, A 0.000, B 0.000, C 0.000 }
gfCNCPoint2[11244] = {X 23.5534, Y 57.7576, Z -3.0000, A 0.000, B 0.000, C 0.000 }
gfCNCPoint2[11245] = {X 21.2879, Y 58.4851, Z -3.0000, A 0.000, B 0.000, C 0.000 }
gfCNCPoint2[11246] = {X 18.9752, Y 59.0448, Z -3.0000, A 0.000, B 0.000, C 0.000 }
gfCNCPoint2[11247] = {X 16.6278, Y 59.4338, Z -3.0000, A 0.000, B 0.000, C 0.000 }
gfCNCPoint2[11248] = {X 14.2583, Y 59.6500, Z -3.0000, A 0.000, B 0.000, C 0.000 }
gfCNCPoint2[11249] = {X 11.8792, Y 59.6923, Z -3.0000, A 0.000, B 0.000, C 0.000 }
gfCNCPoint2[11250] = {X 9.5035, Y 59.5604, Z -3.0000, A 0.000, B 0.000, C 0.000 }
gfCNCPoint2[11251] = {X 9.5035, Y 90.4950, Z -3.0000, A 0.000, B 0.000, C 0.000 }
gfCNCPoint2[11252] = {X 114.8635, Y 90.4950, Z -3.0000, A 0.000, B 0.000, C 0.000 }
gfCNCPoint2[11253] = {X 115.7478, Y 89.2991, Z -3.0000, A 0.000, B 0.000, C 0.000 }
gfCNCPoint2[11254] = {X 116.7724, Y 88.2210, Z -3.0000, A 0.000, B 0.000, C 0.000 }
gfCNCPoint2[11255] = {X 117.9218, Y 87.2769, Z -3.0000, A 0.000, B 0.000, C 0.000 }
gfCNCPoint2[11256] = {X 119.1784, Y 86.4813, Z -3.0000, A 0.000, B 0.000, C 0.000 }
gfCNCPoint2[11257] = {X 120.5233, Y 85.8461, Z -3.0000, A 0.000, B 0.000, C 0.000 }
gfCNCPoint2[11258] = {X 121.9360, Y 85.3810, Z -3.0000, A 0.000, B 0.000, C 0.000 }
gfCNCPoint2[11259] = {X 123.3952, Y 85.0930, Z -3.0000, A 0.000, B 0.000, C 0.000 }
gfCNCPoint2[11260] = {X 123.5620, Y 84.9134, Z -3.0000, A 0.000, B 0.000, C 0.000 }
gfCNCPoint2[11261] = {X 123.7269, Y 84.7321, Z -3.0000, A 0.000, B 0.000, C 0.000 }
gfCNCPoint2[11262] = {X 147.2181, Y 58.9355, Z -3.0000, A 0.000, B 0.000, C 0.000 }
gfCNCPoint2[11263] = {X 147.2180, Y 58.0000, Z -3.0000, A 0.000, B 0.000, C 0.000 }
gfCNCPoint2[11264] = {X 147.2987, Y 56.6058, Z -3.0000, A 0.000, B 0.000, C 0.000 }
gfCNCPoint2[11265] = {X 147.5398, Y 55.2303, Z -3.0000, A 0.000, B 0.000, C 0.000 }
gfCNCPoint2[11266] = {X 148.0022, Y 53.7185, Z -3.0000, A 0.000, B 0.000, C 0.000 }
gfCNCPoint2[11267] = {X 148.6580, Y 52.2800, Z -3.0000, A 0.000, B 0.000, C 0.000 }
gfCNCPoint2[11268] = {X 143.0396, Y 52.2800, Z -3.0000, A 0.000, B 0.000, C 0.000 }
gfCNCPoint2[11269] = {X 141.7807, Y 52.1703, Z -3.0000, A 0.000, B 0.000, C 0.000 }
gfCNCPoint2[11270] = {X 140.5597, Y 51.8446, Z -3.0000, A 0.000, B 0.000, C 0.000 }
gfCNCPoint2[11271] = {X 139.4134, Y 51.3126, Z -3.0000, A 0.000, B 0.000, C 0.000 }
gfCNCPoint2[11272] = {X 138.3764, Y 50.5904, Z -3.0000, A 0.000, B 0.000, C 0.000 }
gfCNCPoint2[11273] = {X 137.4799, Y 49.6998, Z -3.0000, A 0.000, B 0.000, C 0.000 }
gfCNCPoint2[11274] = {X 136.7509, Y 48.6675, Z -3.0000, A 0.000, B 0.000, C 0.000 }
gfCNCPoint2[11275] = {X 136.2114, Y 47.5248, Z -3.0000, A 0.000, B 0.000, C 0.000 }
gfCNCPoint2[11276] = {X 135.8777, Y 46.3059, Z -3.0000, A 0.000, B 0.000, C 0.000 }
gfCNCPoint2[11277] = {X 135.7598, Y 45.0477, Z -3.0000, A 0.000, B 0.000, C 0.000 }
gfCNCPoint2[11278] = {X 135.7601, Y 44.1248, Z -3.0000, A 0.000, B 0.000, C 0.000 }
gfCNCPoint2[11279] = {X 135.8408, Y 43.1249, Z -3.0000, A 0.000, B 0.000, C 0.000 }
gfCNCPoint2[11280] = {X 136.0581, Y 42.1457, Z -3.0000, A 0.000, B 0.000, C 0.000 }
gfCNCPoint2[11281] = {X 138.3597, Y 42.8258, Z -3.0000, A 0.000, B 0.000, C 0.000 }
gfCNCPoint2[11282] = {X 138.6721, Y 42.0319, Z -3.0000, A 0.000, B 0.000, C 0.000 }
gfCNCPoint2[11283] = {X 139.1179, Y 41.3046, Z -3.0000, A 0.000, B 0.000, C 0.000 }
gfCNCPoint2[11284] = {X 139.6836, Y 40.6660, Z -3.0000, A 0.000, B 0.000, C 0.000 }
gfCNCPoint2[11285] = {X 139.6836, Y 20.4368, Z -3.0000, A 0.000, B 0.000, C 0.000 }
gfCNCPoint2[11286] = {X 137.7108, Y 20.4363, Z -3.0000, A 0.000, B 0.000, C 0.000 }
gfCNCPoint2[11287] = {X 137.0003, Y 21.1820, Z -3.0000, A 0.000, B 0.000, C 0.000 }
gfCNCPoint2[11288] = {X 136.1491, Y 21.7619, Z -3.0000, A 0.000, B 0.000, C 0.000 }
gfCNCPoint2[11289] = {X 135.4282, Y 22.0767, Z -3.0000, A 0.000, B 0.000, C 0.000 }
gfCNCPoint2[11290] = {X 134.6660, Y 22.2715, Z -3.0000, A 0.000, B 0.000, C 0.000 }
gfCNCPoint2[11291] = {X 133.8824, Y 22.3414, Z -3.0000, A 0.000, B 0.000, C 0.000 }
gfCNCPoint2[11292] = {X 133.2006, Y 22.3415, Z -3.0000, A 0.000, B 0.000, C 0.000 }
gfCNCPoint2[11293] = {X 132.2486, Y 22.2478, Z -3.0000, A 0.000, B 0.000, C 0.000 }
gfCNCPoint2[11294] = {X 131.3331, Y 21.9701, Z -3.0000, A 0.000, B 0.000, C 0.000 }
gfCNCPoint2[11295] = {X 130.4895, Y 21.5191, Z -3.0000, A 0.000, B 0.000, C 0.000 }
gfCNCPoint2[11296] = {X 129.7500, Y 20.9122, Z -3.0000, A 0.000, B 0.000, C 0.000 }
gfCNCPoint2[11297] = {X 129.1431, Y 20.1727, Z -3.0000, A 0.000, B 0.000, C 0.000 }
gfCNCPoint2[11298] = {X 128.6921, Y 19.3290, Z -3.0000, A 0.000, B 0.000, C 0.000 }
gfCNCPoint2[11299] = {X 128.4144, Y 18.4136, Z -3.0000, A 0.000, B 0.000, C 0.000 }
gfCNCPoint2[11300] = {X 128.3206, Y 17.4615, Z -3.0000, A 0.000, B 0.000, C 0.000 }
gfCNCPoint2[11301] = {X 128.3206, Y 10.4835, Z -3.0000, A 0.000, B 0.000, C 0.000 }
gfCNCPoint2[11302] = {X 128.3317, Y 10.1548, Z -3.0000, A 0.000, B 0.000, C 0.000 }
gfCNCPoint2[11303] = {X 128.3649, Y 9.8276, Z -3.0000, A 0.000, B 0.000, C 0.000 }
gfCNCPoint2[11304] = {X 128.6078, Y 8.8342, Z -3.0000, A 0.000, B 0.000, C 0.000 }
gfCNCPoint2[11305] = {X 129.0524, Y 7.9132, Z -3.0000, A 0.000, B 0.000, C 0.000 }
gfCNCPoint2[11306] = {X 129.6792, Y 7.1050, Z -3.0000, A 0.000, B 0.000, C 0.000 }
gfCNCPoint2[11307] = {X 130.0256, Y 7.4374, Z -3.0000, A 0.000, B 0.000, C 0.000 }
gfCNCPoint2[11308] = {X 130.6996, Y 6.8635, Z -3.0000, A 0.000, B 0.000, C 0.000 }
gfCNCPoint2[11309] = {X 131.4748, Y 6.4361, Z -3.0000, A 0.000, B 0.000, C 0.000 }
gfCNCPoint2[11310] = {X 132.3199, Y 6.1726, Z -3.0000, A 0.000, B 0.000, C 0.000 }
gfCNCPoint2[11311] = {X 133.2007, Y 6.0835, Z -3.0000, A 0.000, B 0.000, C 0.000 }
gfCNCPoint2[11312] = {X 133.8874, Y 6.0837, Z -3.0000, A 0.000, B 0.000, C 0.000 }
gfCNCPoint2[11313] = {X 134.7190, Y 6.1717, Z -3.0000, A 0.000, B 0.000, C 0.000 }
gfCNCPoint2[11314] = {X 135.5189, Y 6.4155, Z -3.0000, A 0.000, B 0.000, C 0.000 }
gfCNCPoint2[11315] = {X 136.2583, Y 6.8061, Z -3.0000, A 0.000, B 0.000, C 0.000 }
gfCNCPoint2[11316] = {X 136.9104, Y 7.3296, Z -3.0000, A 0.000, B 0.000, C 0.000 }
gfCNCPoint2[11317] = {X 137.4516, Y 7.9670, Z -3.0000, A 0.000, B 0.000, C 0.000 }
gfCNCPoint2[11318] = {X 155.0711, Y 7.9670, Z -3.0000, A 0.000, B 0.000, C 0.000 }
gfCNCPoint2[11319] = {X 155.6189, Y 7.3233, Z -3.0000, A 0.000, B 0.000, C 0.000 }
gfCNCPoint2[11320] = {X 156.2796, Y 6.7962, Z -3.0000, A 0.000, B 0.000, C 0.000 }
gfCNCPoint2[11321] = {X 157.0290, Y 6.4052, Z -3.0000, A 0.000, B 0.000, C 0.000 }
gfCNCPoint2[11322] = {X 157.8393, Y 6.1647, Z -3.0000, A 0.000, B 0.000, C 0.000 }
gfCNCPoint2[11323] = {X 158.6806, Y 6.0835, Z -3.0000, A 0.000, B 0.000, C 0.000 }
gfCNCPoint2[11324] = {X 159.3791, Y 6.0839, Z -3.0000, A 0.000, B 0.000, C 0.000 }
gfCNCPoint2[11325] = {X 160.3488, Y 6.2050, Z -3.0000, A 0.000, B 0.000, C 0.000 }
gfCNCPoint2[11326] = {X 161.2678, Y 6.5371, Z -3.0000, A 0.000, B 0.000, C 0.000 }
gfCNCPoint2[11327] = {X 162.0908, Y 7.0639, Z -3.0000, A 0.000, B 0.000, C 0.000 }
gfCNCPoint2[11328] = {X 162.7773, Y 7.7593, Z -3.0000, A 0.000, B 0.000, C 0.000 }
gfCNCPoint2[11329] = {X 163.2934, Y 8.5891, Z -3.0000, A 0.000, B 0.000, C 0.000 }
gfCNCPoint2[11330] = {X 163.6136, Y 9.5124, Z -3.0000, A 0.000, B 0.000, C 0.000 }
gfCNCPoint2[11331] = {X 163.7221, Y 10.4835, Z -3.0000, A 0.000, B 0.000, C 0.000 }
gfCNCPoint2[11332] = {X 163.7221, Y 17.4615, Z -3.0000, A 0.000, B 0.000, C 0.000 }
gfCNCPoint2[11333] = {X 163.6118, Y 18.4406, Z -3.0000, A 0.000, B 0.000, C 0.000 }
gfCNCPoint2[11334] = {X 163.2863, Y 19.3706, Z -3.0000, A 0.000, B 0.000, C 0.000 }
gfCNCPoint2[11335] = {X 162.7621, Y 20.2049, Z -3.0000, A 0.000, B 0.000, C 0.000 }
gfCNCPoint2[11336] = {X 162.0654, Y 20.9016, Z -3.0000, A 0.000, B 0.000, C 0.000 }
gfCNCPoint2[11337] = {X 161.2312, Y 21.4258, Z -3.0000, A 0.000, B 0.000, C 0.000 }
gfCNCPoint2[11338] = {X 160.3012, Y 21.7512, Z -3.0000, A 0.000, B 0.000, C 0.000 }
gfCNCPoint2[11339] = {X 159.3221, Y 21.8615, Z -3.0000, A 0.000, B 0.000, C 0.000 }
gfCNCPoint2[11340] = {X 158.6787, Y 21.8615, Z -3.0000, A 0.000, B 0.000, C 0.000 }
gfCNCPoint2[11341] = {X 157.8333, Y 21.7762, Z -3.0000, A 0.000, B 0.000, C 0.000 }
gfCNCPoint2[11342] = {X 157.0197, Y 21.5314, Z -3.0000, A 0.000, B 0.000, C 0.000 }
gfCNCPoint2[11343] = {X 156.2677, Y 21.1360, Z -3.0000, A 0.000, B 0.000, C 0.000 }
gfCNCPoint2[11344] = {X 155.6048, Y 20.6044, Z -3.0000, A 0.000, B 0.000, C 0.000 }
gfCNCPoint2[11345] = {X 155.0554, Y 19.9563, Z -3.0000, A 0.000, B 0.000, C 0.000 }
gfCNCPoint2[11346] = {X 152.3560, Y 19.9576, Z -3.0000, A 0.000, B 0.000, C 0.000 }
gfCNCPoint2[11347] = {X 152.3544, Y 40.8428, Z -3.0000, A 0.000, B 0.000, C 0.000 }
gfCNCPoint2[11348] = {X 152.8075, Y 41.3313, Z -3.0000, A 0.000, B 0.000, C 0.000 }
gfCNCPoint2[11349] = {X 152.8994, Y 41.4411, Z -3.0000, A 0.000, B 0.000, C 0.000 }
gfCNCPoint2[11350] = {X 153.4337, Y 42.2815, Z -3.0000, A 0.000, B 0.000, C 0.000 }
gfCNCPoint2[11351] = {X 153.7672, Y 43.2198, Z -3.0000, A 0.000, B 0.000, C 0.000 }
gfCNCPoint2[11352] = {X 153.8831, Y 44.2089, Z -3.0000, A 0.000, B 0.000, C 0.000 }
gfCNCPoint2[11353] = {X 153.8829, Y 45.0423, Z -3.0000, A 0.000, B 0.000, C 0.000 }
gfCNCPoint2[11354] = {X 153.7646, Y 46.0144, Z -3.0000, A 0.000, B 0.000, C 0.000 }
gfCNCPoint2[11355] = {X 153.4342, Y 46.9363, Z -3.0000, A 0.000, B 0.000, C 0.000 }
gfCNCPoint2[11356] = {X 152.9080, Y 47.7622, Z -3.0000, A 0.000, B 0.000, C 0.000 }
gfCNCPoint2[11357] = {X 152.2123, Y 48.4513, Z -3.0000, A 0.000, B 0.000, C 0.000 }
gfCNCPoint2[11358] = {X 151.3813, Y 48.9695, Z -3.0000, A 0.000, B 0.000, C 0.000 }
gfCNCPoint2[11359] = {X 150.4563, Y 49.2910, Z -3.0000, A 0.000, B 0.000, C 0.000 }
gfCNCPoint2[11360] = {X 149.4831, Y 49.4000, Z -3.0000, A 0.000, B 0.000, C 0.000 }
gfCNCPoint2[11361] = {X 143.0396, Y 49.4000, Z -3.0000, A 0.000, B 0.000, C 0.000 }
gfCNCPoint2[11362] = {X 142.0605, Y 49.2897, Z -3.0000, A 0.000, B 0.000, C 0.000 }
gfCNCPoint2[11363] = {X 141.1305, Y 48.9643, Z -3.0000, A 0.000, B 0.000, C 0.000 }
gfCNCPoint2[11364] = {X 140.2963, Y 48.4400, Z -3.0000, A 0.000, B 0.000, C 0.000 }
gfCNCPoint2[11365] = {X 139.5996, Y 47.7433, Z -3.0000, A 0.000, B 0.000, C 0.000 }
gfCNCPoint2[11366] = {X 139.0754, Y 46.9091, Z -3.0000, A 0.000, B 0.000, C 0.000 }
gfCNCPoint2[11367] = {X 138.7499, Y 45.9791, Z -3.0000, A 0.000, B 0.000, C 0.000 }
gfCNCPoint2[11368] = {X 138.6396, Y 45.0000, Z -3.0000, A 0.000, B 0.000, C 0.000 }
gfCNCPoint2[11369] = {X 138.6400, Y 44.1483, Z -3.0000, A 0.000, B 0.000, C 0.000 }
gfCNCPoint2[11370] = {X 138.7505, Y 43.2275, Z -3.0000, A 0.000, B 0.000, C 0.000 }
gfCNCPoint2[11371] = {X 139.0514, Y 42.3503, Z -3.0000, A 0.000, B 0.000, C 0.000 }
gfCNCPoint2[11372] = {X 139.5295, Y 41.5556, Z -3.0000, A 0.000, B 0.000, C 0.000 }
gfCNCPoint2[11373] = {X 140.1636, Y 40.8789, Z -3.0000, A 0.000, B 0.000, C 0.000 }
gfCNCPoint2[11374] = {X 140.1636, Y 19.9570, Z -3.0000, A 0.000, B 0.000, C 0.000 }
gfCNCPoint2[11375] = {X 137.4667, Y 19.9563, Z -3.0000, A 0.000, B 0.000, C 0.000 }
gfCNCPoint2[11376] = {X 136.9191, Y 20.6070, Z -3.0000, A 0.000, B 0.000, C 0.000 }
gfCNCPoint2[11377] = {X 136.2564, Y 21.1401, Z -3.0000, A 0.000, B 0.000, C 0.000 }
gfCNCPoint2[11378] = {X 135.5036, Y 21.5359, Z -3.0000, A 0.000, B 0.000, C 0.000 }
gfCNCPoint2[11379] = {X 134.6887, Y 21.7794, Z -3.0000, A 0.000, B 0.000, C 0.000 }
gfCNCPoint2[11380] = {X 133.8421, Y 21.8615, Z -3.0000, A 0.000, B 0.000, C 0.000 }
gfCNCPoint2[11381] = {X 133.2006, Y 21.8615, Z -3.0000, A 0.000, B 0.000, C 0.000 }
gfCNCPoint2[11382] = {X 132.2215, Y 21.7512, Z -3.0000, A 0.000, B 0.000, C 0.000 }
gfCNCPoint2[11383] = {X 131.2916, Y 21.4258, Z -3.0000, A 0.000, B 0.000, C 0.000 }
gfCNCPoint2[11384] = {X 130.4573, Y 20.9016, Z -3.0000, A 0.000, B 0.000, C 0.000 }
gfCNCPoint2[11385] = {X 129.7606, Y 20.2049, Z -3.0000, A 0.000, B 0.000, C 0.000 }
gfCNCPoint2[11386] = {X 129.2364, Y 19.3706, Z -3.0000, A 0.000, B 0.000, C 0.000 }
gfCNCPoint2[11387] = {X 128.9110, Y 18.4406, Z -3.0000, A 0.000, B 0.000, C 0.000 }
gfCNCPoint2[11388] = {X 128.8006, Y 17.4615, Z -3.0000, A 0.000, B 0.000, C 0.000 }
gfCNCPoint2[11389] = {X 128.8006, Y 10.4835, Z -3.0000, A 0.000, B 0.000, C 0.000 }
gfCNCPoint2[11390] = {X 128.8808, Y 9.6475, Z -3.0000, A 0.000, B 0.000, C 0.000 }
gfCNCPoint2[11391] = {X 129.1184, Y 8.8419, Z -3.0000, A 0.000, B 0.000, C 0.000 }
gfCNCPoint2[11392] = {X 129.5046, Y 8.0961, Z -3.0000, A 0.000, B 0.000, C 0.000 }
gfCNCPoint2[11393] = {X 130.0256, Y 7.4374, Z -3.0000, A 0.000, B 0.000, C 0.000 }
gfCNCPoint2[11394] = {X 129.6792, Y 7.1050, Z -3.0000, A 0.000, B 0.000, C 0.000 }
gfCNCPoint2[11395] = {X 102.4337, Y 7.1050, Z -3.0000, A 0.000, B 0.000, C 0.000 }
gfCNCPoint2[11396] = {X 102.4337, Y 11.9050, Z -3.0000, A 0.000, B 0.000, C 0.000 }
gfCNCPoint2[11397] = {X 101.3242, Y 11.9050, Z -3.0000, A 0.000, B 0.000, C 0.000 }
gfCNCPoint2[11398] = {X 101.3283, Y 12.0459, Z -3.0000, A 0.000, B 0.000, C 0.000 }
gfCNCPoint2[11399] = {X 101.3297, Y 12.1868, Z -3.0000, A 0.000, B 0.000, C 0.000 }
gfCNCPoint2[11400] = {X 101.3293, Y 13.0462, Z -3.0000, A 0.000, B 0.000, C 0.000 }
gfCNCPoint2[11401] = {X 101.2274, Y 14.1941, Z -3.0000, A 0.000, B 0.000, C 0.000 }
gfCNCPoint2[11402] = {X 100.9455, Y 15.3116, Z -3.0000, A 0.000, B 0.000, C 0.000 }
gfCNCPoint2[11403] = {X 101.0390, Y 15.5442, Z -3.0000, A 0.000, B 0.000, C 0.000 }
gfCNCPoint2[11404] = {X 101.8684, Y 17.6003, Z -3.0000, A 0.000, B 0.000, C 0.000 }
gfCNCPoint2[11405] = {X 102.8004, Y 15.2759, Z -3.0000, A 0.000, B 0.000, C 0.000 }
gfCNCPoint2[11406] = {X 102.5274, Y 14.1752, Z -3.0000, A 0.000, B 0.000, C 0.000 }
gfCNCPoint2[11407] = {X 102.4286, Y 13.0454, Z -3.0000, A 0.000, B 0.000, C 0.000 }
gfCNCPoint2[11408] = {X 102.4283, Y 12.1868, Z -3.0000, A 0.000, B 0.000, C 0.000 }
gfCNCPoint2[11409] = {X 102.4296, Y 12.0459, Z -3.0000, A 0.000, B 0.000, C 0.000 }
gfCNCPoint2[11410] = {X 102.4337, Y 11.9050, Z -3.0000, A 0.000, B 0.000, C 0.000 }
gfCNCPoint2[11411] = {X 102.4337, Y 9.5050, Z -3.0000, A 0.000, B 0.000, C 0.000 }
gfCNCPoint2[11412] = {X 98.1267, Y 9.5050, Z -3.0000, A 0.000, B 0.000, C 0.000 }
gfCNCPoint2[11413] = {X 98.5430, Y 10.2829, Z -3.0000, A 0.000, B 0.000, C 0.000 }
gfCNCPoint2[11414] = {X 98.8123, Y 11.1230, Z -3.0000, A 0.000, B 0.000, C 0.000 }
gfCNCPoint2[11415] = {X 98.9260, Y 11.9979, Z -3.0000, A 0.000, B 0.000, C 0.000 }
gfCNCPoint2[11416] = {X 98.9288, Y 12.0924, Z -3.0000, A 0.000, B 0.000, C 0.000 }
gfCNCPoint2[11417] = {X 98.9297, Y 12.1868, Z -3.0000, A 0.000, B 0.000, C 0.000 }
gfCNCPoint2[11418] = {X 98.9294, Y 13.0237, Z -3.0000, A 0.000, B 0.000, C 0.000 }
gfCNCPoint2[11419] = {X 98.8589, Y 13.8060, Z -3.0000, A 0.000, B 0.000, C 0.000 }
gfCNCPoint2[11420] = {X 98.6638, Y 14.5668, Z -3.0000, A 0.000, B 0.000, C 0.000 }
gfCNCPoint2[11421] = {X 98.3491, Y 15.2865, Z -3.0000, A 0.000, B 0.000, C 0.000 }
gfCNCPoint2[11422] = {X 98.8126, Y 16.4404, Z -3.0000, A 0.000, B 0.000, C 0.000 }
gfCNCPoint2[11423] = {X 101.8752, Y 24.0320, Z -3.0000, A 0.000, B 0.000, C 0.000 }
gfCNCPoint2[11424] = {X 105.3935, Y 15.2577, Z -3.0000, A 0.000, B 0.000, C 0.000 }
gfCNCPoint2[11425] = {X 105.0871, Y 14.5461, Z -3.0000, A 0.000, B 0.000, C 0.000 }
gfCNCPoint2[11426] = {X 104.8971, Y 13.7949, Z -3.0000, A 0.000, B 0.000, C 0.000 }
gfCNCPoint2[11427] = {X 104.8285, Y 13.0231, Z -3.0000, A 0.000, B 0.000, C 0.000 }
gfCNCPoint2[11428] = {X 104.8283, Y 12.1868, Z -3.0000, A 0.000, B 0.000, C 0.000 }
gfCNCPoint2[11429] = {X 104.8292, Y 12.0924, Z -3.0000, A 0.000, B 0.000, C 0.000 }
gfCNCPoint2[11430] = {X 104.8319, Y 11.9979, Z -3.0000, A 0.000, B 0.000, C 0.000 }
gfCNCPoint2[11431] = {X 104.9456, Y 11.1230, Z -3.0000, A 0.000, B 0.000, C 0.000 }
gfCNCPoint2[11432] = {X 105.2150, Y 10.2829, Z -3.0000, A 0.000, B 0.000, C 0.000 }
gfCNCPoint2[11433] = {X 105.6312, Y 9.5050, Z -3.0000, A 0.000, B 0.000, C 0.000 }
gfCNCPoint2[11434] = {X 102.4337, Y 9.5050, Z -3.0000, A 0.000, B 0.000, C 0.000 }
gfCNCPoint2[11435] = {X 102.4337, Y 7.1050, Z -3.0000, A 0.000, B 0.000, C 0.000 }
gfCNCPoint2[11436] = {X 64.8350, Y 7.1050, Z -3.0000, A 0.000, B 0.000, C 0.000 }
gfCNCPoint2[11437] = {X 65.5947, Y 8.0242, Z -3.0000, A 0.000, B 0.000, C 0.000 }
gfCNCPoint2[11438] = {X 66.1941, Y 9.0551, Z -3.0000, A 0.000, B 0.000, C 0.000 }
gfCNCPoint2[11439] = {X 66.6172, Y 10.1699, Z -3.0000, A 0.000, B 0.000, C 0.000 }
gfCNCPoint2[11440] = {X 66.8305, Y 11.1684, Z -3.0000, A 0.000, B 0.000, C 0.000 }
gfCNCPoint2[11441] = {X 66.9021, Y 12.1868, Z -3.0000, A 0.000, B 0.000, C 0.000 }
gfCNCPoint2[11442] = {X 66.9018, Y 13.0462, Z -3.0000, A 0.000, B 0.000, C 0.000 }
gfCNCPoint2[11443] = {X 66.7771, Y 14.3213, Z -3.0000, A 0.000, B 0.000, C 0.000 }
gfCNCPoint2[11444] = {X 66.4309, Y 15.5548, Z -3.0000, A 0.000, B 0.000, C 0.000 }
gfCNCPoint2[11445] = {X 74.9107, Y 38.2388, Z -3.0000, A 0.000, B 0.000, C 0.000 }
gfCNCPoint2[11446] = {X 75.8032, Y 38.9736, Z -3.0000, A 0.000, B 0.000, C 0.000 }
gfCNCPoint2[11447] = {X 76.5682, Y 39.8404, Z -3.0000, A 0.000, B 0.000, C 0.000 }
gfCNCPoint2[11448] = {X 77.1863, Y 40.8174, Z -3.0000, A 0.000, B 0.000, C 0.000 }
gfCNCPoint2[11449] = {X 77.6419, Y 41.8798, Z -3.0000, A 0.000, B 0.000, C 0.000 }
gfCNCPoint2[11450] = {X 77.9236, Y 43.0011, Z -3.0000, A 0.000, B 0.000, C 0.000 }
gfCNCPoint2[11451] = {X 78.0243, Y 44.1527, Z -3.0000, A 0.000, B 0.000, C 0.000 }
gfCNCPoint2[11452] = {X 78.0245, Y 45.0000, Z -3.0000, A 0.000, B 0.000, C 0.000 }
gfCNCPoint2[11453] = {X 77.9139, Y 46.2642, Z -3.0000, A 0.000, B 0.000, C 0.000 }
gfCNCPoint2[11454] = {X 77.5854, Y 47.4899, Z -3.0000, A 0.000, B 0.000, C 0.000 }
gfCNCPoint2[11455] = {X 77.0491, Y 48.6400, Z -3.0000, A 0.000, B 0.000, C 0.000 }
gfCNCPoint2[11456] = {X 76.3213, Y 49.6795, Z -3.0000, A 0.000, B 0.000, C 0.000 }
gfCNCPoint2[11457] = {X 75.4240, Y 50.5768, Z -3.0000, A 0.000, B 0.000, C 0.000 }
gfCNCPoint2[11458] = {X 74.3845, Y 51.3047, Z -3.0000, A 0.000, B 0.000, C 0.000 }
gfCNCPoint2[11459] = {X 73.2344, Y 51.8410, Z -3.0000, A 0.000, B 0.000, C 0.000 }
gfCNCPoint2[11460] = {X 72.0086, Y 52.1694, Z -3.0000, A 0.000, B 0.000, C 0.000 }
gfCNCPoint2[11461] = {X 70.7445, Y 52.2800, Z -3.0000, A 0.000, B 0.000, C 0.000 }
gfCNCPoint2[11462] = {X 64.1851, Y 52.2800, Z -3.0000, A 0.000, B 0.000, C 0.000 }
gfCNCPoint2[11463] = {X 62.9397, Y 52.1727, Z -3.0000, A 0.000, B 0.000, C 0.000 }
gfCNCPoint2[11464] = {X 61.7311, Y 51.8539, Z -3.0000, A 0.000, B 0.000, C 0.000 }
gfCNCPoint2[11465] = {X 60.5947, Y 51.3330, Z -3.0000, A 0.000, B 0.000, C 0.000 }
gfCNCPoint2[11466] = {X 59.5643, Y 50.6255, Z -3.0000, A 0.000, B 0.000, C 0.000 }
gfCNCPoint2[11467] = {X 58.6700, Y 49.7521, Z -3.0000, A 0.000, B 0.000, C 0.000 }
gfCNCPoint2[11468] = {X 57.9384, Y 48.7385, Z -3.0000, A 0.000, B 0.000, C 0.000 }
gfCNCPoint2[11469] = {X 57.3706, Y 47.5614, Z -3.0000, A 0.000, B 0.000, C 0.000 }
gfCNCPoint2[11470] = {X 57.0224, Y 46.3017, Z -3.0000, A 0.000, B 0.000, C 0.000 }
gfCNCPoint2[11471] = {X 56.9051, Y 45.0000, Z -3.0000, A 0.000, B 0.000, C 0.000 }
gfCNCPoint2[11472] = {X 56.9052, Y 44.1968, Z -3.0000, A 0.000, B 0.000, C 0.000 }
gfCNCPoint2[11473] = {X 56.9289, Y 43.6212, Z -3.0000, A 0.000, B 0.000, C 0.000 }
gfCNCPoint2[11474] = {X 56.9981, Y 43.0492, Z -3.0000, A 0.000, B 0.000, C 0.000 }
gfCNCPoint2[11475] = {X 54.7600, Y 43.0492, Z -3.0000, A 0.000, B 0.000, C 0.000 }
gfCNCPoint2[11476] = {X 54.8275, Y 43.6012, Z -3.0000, A 0.000, B 0.000, C 0.000 }
gfCNCPoint2[11477] = {X 54.8528, Y 44.1567, Z -3.0000, A 0.000, B 0.000, C 0.000 }
gfCNCPoint2[11478] = {X 54.8529, Y 45.0000, Z -3.0000, A 0.000, B 0.000, C 0.000 }
gfCNCPoint2[11479] = {X 54.7356, Y 46.3017, Z -3.0000, A 0.000, B 0.000, C 0.000 }
gfCNCPoint2[11480] = {X 54.3875, Y 47.5614, Z -3.0000, A 0.000, B 0.000, C 0.000 }
gfCNCPoint2[11481] = {X 53.8197, Y 48.7385, Z -3.0000, A 0.000, B 0.000, C 0.000 }
gfCNCPoint2[11482] = {X 53.0880, Y 49.7521, Z -3.0000, A 0.000, B 0.000, C 0.000 }
gfCNCPoint2[11483] = {X 52.1938, Y 50.6255, Z -3.0000, A 0.000, B 0.000, C 0.000 }
gfCNCPoint2[11484] = {X 51.1633, Y 51.3330, Z -3.0000, A 0.000, B 0.000, C 0.000 }
gfCNCPoint2[11485] = {X 50.0270, Y 51.8539, Z -3.0000, A 0.000, B 0.000, C 0.000 }
gfCNCPoint2[11486] = {X 48.8183, Y 52.1727, Z -3.0000, A 0.000, B 0.000, C 0.000 }
gfCNCPoint2[11487] = {X 47.5729, Y 52.2800, Z -3.0000, A 0.000, B 0.000, C 0.000 }
gfCNCPoint2[11488] = {X 40.6393, Y 52.2800, Z -3.0000, A 0.000, B 0.000, C 0.000 }
gfCNCPoint2[11489] = {X 39.4476, Y 52.1818, Z -3.0000, A 0.000, B 0.000, C 0.000 }
gfCNCPoint2[11490] = {X 38.2881, Y 51.8899, Z -3.0000, A 0.000, B 0.000, C 0.000 }
gfCNCPoint2[11491] = {X 37.1919, Y 51.4120, Z -3.0000, A 0.000, B 0.000, C 0.000 }
gfCNCPoint2[11492] = {X 36.1888, Y 50.7612, Z -3.0000, A 0.000, B 0.000, C 0.000 }
gfCNCPoint2[11493] = {X 35.3058, Y 49.9550, Z -3.0000, A 0.000, B 0.000, C 0.000 }
gfCNCPoint2[11494] = {X 34.8234, Y 50.4196, Z -3.0000, A 0.000, B 0.000, C 0.000 }
gfCNCPoint2[11495] = {X 34.3150, Y 50.8555, Z -3.0000, A 0.000, B 0.000, C 0.000 }
gfCNCPoint2[11496] = {X 33.7728, Y 51.2939, Z -3.0000, A 0.000, B 0.000, C 0.000 }
gfCNCPoint2[11497] = {X 32.5155, Y 52.1777, Z -3.0000, A 0.000, B 0.000, C 0.000 }
gfCNCPoint2[11498] = {X 31.1525, Y 52.8878, Z -3.0000, A 0.000, B 0.000, C 0.000 }
gfCNCPoint2[11499] = {X 29.7077, Y 53.4117, Z -3.0000, A 0.000, B 0.000, C 0.000 }
gfCNCPoint2[11500] = {X 28.2064, Y 53.7404, Z -3.0000, A 0.000, B 0.000, C 0.000 }
gfCNCPoint2[11501] = {X 26.6748, Y 53.8680, Z -3.0000, A 0.000, B 0.000, C 0.000 }
gfCNCPoint2[11502] = {X 24.7380, Y 54.7407, Z -3.0000, A 0.000, B 0.000, C 0.000 }
gfCNCPoint2[11503] = {X 22.7521, Y 55.4953, Z -3.0000, A 0.000, B 0.000, C 0.000 }
gfCNCPoint2[11504] = {X 20.2259, Y 56.2874, Z -3.0000, A 0.000, B 0.000, C 0.000 }
gfCNCPoint2[11505] = {X 17.6398, Y 56.8545, Z -3.0000, A 0.000, B 0.000, C 0.000 }
gfCNCPoint2[11506] = {X 15.0140, Y 57.1922, Z -3.0000, A 0.000, B 0.000, C 0.000 }
gfCNCPoint2[11507] = {X 12.3686, Y 57.2978, Z -3.0000, A 0.000, B 0.000, C 0.000 }
gfCNCPoint2[11508] = {X 9.7242, Y 57.1706, Z -3.0000, A 0.000, B 0.000, C 0.000 }
gfCNCPoint2[11509] = {X 8.4099, Y 57.0201, Z -3.0000, A 0.000, B 0.000, C 0.000 }
gfCNCPoint2[11510] = {X 7.1035, Y 56.8120, Z -3.0000, A 0.000, B 0.000, C 0.000 }
gfCNCPoint2[11511] = {X 7.1035, Y 92.8950, Z -3.0000, A 0.000, B 0.000, C 0.000 }
gfCNCPoint2[11512] = {X 116.2647, Y 92.8950, Z -3.0000, A 0.000, B 0.000, C 0.000 }
gfCNCPoint2[11513] = {X 116.9724, Y 91.6566, Z -3.0000, A 0.000, B 0.000, C 0.000 }
gfCNCPoint2[11514] = {X 117.8544, Y 90.5358, Z -3.0000, A 0.000, B 0.000, C 0.000 }
gfCNCPoint2[11515] = {X 118.8915, Y 89.5567, Z -3.0000, A 0.000, B 0.000, C 0.000 }
gfCNCPoint2[11516] = {X 120.0613, Y 88.7406, Z -3.0000, A 0.000, B 0.000, C 0.000 }
gfCNCPoint2[11517] = {X 121.3382, Y 88.1053, Z -3.0000, A 0.000, B 0.000, C 0.000 }
gfCNCPoint2[11518] = {X 122.6947, Y 87.6645, Z -3.0000, A 0.000, B 0.000, C 0.000 }
gfCNCPoint2[11519] = {X 124.1012, Y 87.4278, Z -3.0000, A 0.000, B 0.000, C 0.000 }
gfCNCPoint2[11520] = {X 124.5364, Y 87.3622, Z -3.0000, A 0.000, B 0.000, C 0.000 }
gfCNCPoint2[11521] = {X 125.0282, Y 86.8592, Z -3.0000, A 0.000, B 0.000, C 0.000 }
gfCNCPoint2[11522] = {X 125.5060, Y 86.3430, Z -3.0000, A 0.000, B 0.000, C 0.000 }
gfCNCPoint2[11523] = {X 149.6586, Y 59.8200, Z -3.0000, A 0.000, B 0.000, C 0.000 }
gfCNCPoint2[11524] = {X 149.6295, Y 59.4070, Z -3.0000, A 0.000, B 0.000, C 0.000 }
gfCNCPoint2[11525] = {X 149.6181, Y 58.9930, Z -3.0000, A 0.000, B 0.000, C 0.000 }
gfCNCPoint2[11526] = {X 149.6180, Y 58.0000, Z -3.0000, A 0.000, B 0.000, C 0.000 }
gfCNCPoint2[11527] = {X 149.6915, Y 56.8093, Z -3.0000, A 0.000, B 0.000, C 0.000 }
gfCNCPoint2[11528] = {X 149.9109, Y 55.6367, Z -3.0000, A 0.000, B 0.000, C 0.000 }
gfCNCPoint2[11529] = {X 150.2729, Y 54.5000, Z -3.0000, A 0.000, B 0.000, C 0.000 }
gfCNCPoint2[11530] = {X 150.7719, Y 53.4164, Z -3.0000, A 0.000, B 0.000, C 0.000 }
gfCNCPoint2[11531] = {X 151.5117, Y 52.2488, Z -3.0000, A 0.000, B 0.000, C 0.000 }
gfCNCPoint2[11532] = {X 152.4103, Y 51.1984, Z -3.0000, A 0.000, B 0.000, C 0.000 }
gfCNCPoint2[11533] = {X 153.4493, Y 50.2867, Z -3.0000, A 0.000, B 0.000, C 0.000 }
gfCNCPoint2[11534] = {X 154.6075, Y 49.5323, Z -3.0000, A 0.000, B 0.000, C 0.000 }
gfCNCPoint2[11535] = {X 155.8614, Y 48.9505, Z -3.0000, A 0.000, B 0.000, C 0.000 }
gfCNCPoint2[11536] = {X 157.1854, Y 48.5533, Z -3.0000, A 0.000, B 0.000, C 0.000 }
gfCNCPoint2[11537] = {X 158.2353, Y 48.3785, Z -3.0000, A 0.000, B 0.000, C 0.000 }
gfCNCPoint2[11538] = {X 159.2980, Y 48.3200, Z -3.0000, A 0.000, B 0.000, C 0.000 }
gfCNCPoint2[11539] = {X 176.3110, Y 48.3200, Z -3.0000, A 0.000, B 0.000, C 0.000 }
gfCNCPoint2[11540] = {X 175.1963, Y 47.6606, Z -3.0000, A 0.000, B 0.000, C 0.000 }
gfCNCPoint2[11541] = {X 174.1331, Y 46.9211, Z -3.0000, A 0.000, B 0.000, C 0.000 }
gfCNCPoint2[11542] = {X 172.7674, Y 45.7586, Z -3.0000, A 0.000, B 0.000, C 0.000 }
gfCNCPoint2[11543] = {X 171.5641, Y 44.4288, Z -3.0000, A 0.000, B 0.000, C 0.000 }
gfCNCPoint2[11544] = {X 170.6261, Y 43.0901, Z -3.0000, A 0.000, B 0.000, C 0.000 }
gfCNCPoint2[11545] = {X 169.8531, Y 41.6499, Z -3.0000, A 0.000, B 0.000, C 0.000 }
gfCNCPoint2[11546] = {X 169.2558, Y 40.1283, Z -3.0000, A 0.000, B 0.000, C 0.000 }
gfCNCPoint2[11547] = {X 168.8427, Y 38.5468, Z -3.0000, A 0.000, B 0.000, C 0.000 }
gfCNCPoint2[11548] = {X 168.6196, Y 36.9275, Z -3.0000, A 0.000, B 0.000, C 0.000 }
gfCNCPoint2[11549] = {X 168.5333, Y 35.0260, Z -3.0000, A 0.000, B 0.000, C 0.000 }
gfCNCPoint2[11550] = {X 168.6855, Y 33.1286, Z -3.0000, A 0.000, B 0.000, C 0.000 }
gfCNCPoint2[11551] = {X 169.0736, Y 31.2651, Z -3.0000, A 0.000, B 0.000, C 0.000 }
gfCNCPoint2[11552] = {X 169.6918, Y 29.4647, Z -3.0000, A 0.000, B 0.000, C 0.000 }
gfCNCPoint2[11553] = {X 170.2639, Y 28.2680, Z -3.0000, A 0.000, B 0.000, C 0.000 }
gfCNCPoint2[11554] = {X 170.9709, Y 27.1457, Z -3.0000, A 0.000, B 0.000, C 0.000 }
gfCNCPoint2[11555] = {X 171.8033, Y 26.1129, Z -3.0000, A 0.000, B 0.000, C 0.000 }
gfCNCPoint2[11556] = {X 172.7497, Y 25.1835, Z -3.0000, A 0.000, B 0.000, C 0.000 }
gfCNCPoint2[11557] = {X 173.7976, Y 24.3702, Z -3.0000, A 0.000, B 0.000, C 0.000 }
gfCNCPoint2[11558] = {X 173.0272, Y 23.7519, Z -3.0000, A 0.000, B 0.000, C 0.000 }
gfCNCPoint2[11559] = {X 172.3972, Y 22.9912, Z -3.0000, A 0.000, B 0.000, C 0.000 }
gfCNCPoint2[11560] = {X 171.9332, Y 22.1192, Z -3.0000, A 0.000, B 0.000, C 0.000 }
gfCNCPoint2[11561] = {X 169.3220, Y 15.7237, Z -3.0000, A 0.000, B 0.000, C 0.000 }
gfCNCPoint2[11562] = {X 169.1088, Y 15.0753, Z -3.0000, A 0.000, B 0.000, C 0.000 }
gfCNCPoint2[11563] = {X 168.9882, Y 14.4035, Z -3.0000, A 0.000, B 0.000, C 0.000 }
gfCNCPoint2[11564] = {X 168.9599, Y 13.8791, Z -3.0000, A 0.000, B 0.000, C 0.000 }
gfCNCPoint2[11565] = {X 168.9882, Y 13.3548, Z -3.0000, A 0.000, B 0.000, C 0.000 }
gfCNCPoint2[11566] = {X 169.1590, Y 12.4995, Z -3.0000, A 0.000, B 0.000, C 0.000 }
gfCNCPoint2[11567] = {X 169.4794, Y 11.6883, Z -3.0000, A 0.000, B 0.000, C 0.000 }
gfCNCPoint2[11568] = {X 169.9390, Y 10.9470, Z -3.0000, A 0.000, B 0.000, C 0.000 }
gfCNCPoint2[11569] = {X 170.6134, Y 10.2180, Z -3.0000, A 0.000, B 0.000, C 0.000 }
gfCNCPoint2[11570] = {X 171.4215, Y 9.6405, Z -3.0000, A 0.000, B 0.000, C 0.000 }
gfCNCPoint2[11571] = {X 172.0576, Y 9.2779, Z -3.0000, A 0.000, B 0.000, C 0.000 }
gfCNCPoint2[11572] = {X 172.9937, Y 8.8768, Z -3.0000, A 0.000, B 0.000, C 0.000 }
gfCNCPoint2[11573] = {X 173.9927, Y 8.6787, Z -3.0000, A 0.000, B 0.000, C 0.000 }
gfCNCPoint2[11574] = {X 175.0111, Y 8.6923, Z -3.0000, A 0.000, B 0.000, C 0.000 }
gfCNCPoint2[11575] = {X 176.0044, Y 8.9170, Z -3.0000, A 0.000, B 0.000, C 0.000 }
gfCNCPoint2[11576] = {X 177.7787, Y 8.1690, Z -3.0000, A 0.000, B 0.000, C 0.000 }
gfCNCPoint2[11577] = {X 179.6066, Y 7.5638, Z -3.0000, A 0.000, B 0.000, C 0.000 }
gfCNCPoint2[11578] = {X 181.4766, Y 7.1050, Z -3.0000, A 0.000, B 0.000, C 0.000 }
gfCNCPoint2[11579] = {X 168.0205, Y 7.1050, Z -3.0000, A 0.000, B 0.000, C 0.000 }
gfCNCPoint2[11580] = {X 168.0205, Y 4.7050, Z -3.0000, A 0.000, B 0.000, C 0.000 }
gfCNCPoint2[11581] = {X 155.1590, Y 4.7050, Z -3.0000, A 0.000, B 0.000, C 0.000 }
gfCNCPoint2[11582] = {X 155.1590, Y 7.1050, Z -3.0000, A 0.000, B 0.000, C 0.000 }
gfCNCPoint2[11583] = {X 137.3637, Y 7.1050, Z -3.0000, A 0.000, B 0.000, C 0.000 }
gfCNCPoint2[11584] = {X 137.5338, Y 7.2918, Z -3.0000, A 0.000, B 0.000, C 0.000 }
gfCNCPoint2[11585] = {X 137.6940, Y 7.4870, Z -3.0000, A 0.000, B 0.000, C 0.000 }
gfCNCPoint2[11586] = {X 154.8287, Y 7.4870, Z -3.0000, A 0.000, B 0.000, C 0.000 }
gfCNCPoint2[11587] = {X 154.9889, Y 7.2918, Z -3.0000, A 0.000, B 0.000, C 0.000 }
gfCNCPoint2[11588] = {X 155.1590, Y 7.1050, Z -3.0000, A 0.000, B 0.000, C 0.000 }
gfCNCPoint2[11589] = {X 155.1590, Y 4.7050, Z -3.0000, A 0.000, B 0.000, C 0.000 }
gfCNCPoint2[11590] = {X 42.6031, Y 4.7050, Z -3.0000, A 0.000, B 0.000, C 0.000 }
gfCNCPoint2[11591] = {X 42.6031, Y 9.5050, Z -3.0000, A 0.000, B 0.000, C 0.000 }
gfCNCPoint2[11592] = {X 36.0453, Y 9.5050, Z -3.0000, A 0.000, B 0.000, C 0.000 }
gfCNCPoint2[11593] = {X 37.0554, Y 11.3888, Z -3.0000, A 0.000, B 0.000, C 0.000 }
gfCNCPoint2[11594] = {X 37.8837, Y 13.3593, Z -3.0000, A 0.000, B 0.000, C 0.000 }
gfCNCPoint2[11595] = {X 38.5463, Y 15.5415, Z -3.0000, A 0.000, B 0.000, C 0.000 }
gfCNCPoint2[11596] = {X 39.0047, Y 17.7755, Z -3.0000, A 0.000, B 0.000, C 0.000 }
gfCNCPoint2[11597] = {X 39.2551, Y 20.0424, Z -3.0000, A 0.000, B 0.000, C 0.000 }
gfCNCPoint2[11598] = {X 39.2951, Y 22.3226, Z -3.0000, A 0.000, B 0.000, C 0.000 }
gfCNCPoint2[11599] = {X 39.1246, Y 24.5968, Z -3.0000, A 0.000, B 0.000, C 0.000 }
gfCNCPoint2[11600] = {X 42.5394, Y 15.4281, Z -3.0000, A 0.000, B 0.000, C 0.000 }
gfCNCPoint2[11601] = {X 42.3075, Y 14.2453, Z -3.0000, A 0.000, B 0.000, C 0.000 }
gfCNCPoint2[11602] = {X 42.2244, Y 13.0428, Z -3.0000, A 0.000, B 0.000, C 0.000 }
gfCNCPoint2[11603] = {X 42.2242, Y 12.1868, Z -3.0000, A 0.000, B 0.000, C 0.000 }
gfCNCPoint2[11604] = {X 42.3194, Y 10.8326, Z -3.0000, A 0.000, B 0.000, C 0.000 }
gfCNCPoint2[11605] = {X 42.6031, Y 9.5050, Z -3.0000, A 0.000, B 0.000, C 0.000 }
gfCNCPoint2[11606] = {X 42.6031, Y 7.1050, Z -3.0000, A 0.000, B 0.000, C 0.000 }
gfCNCPoint2[11607] = {X 31.2108, Y 7.1050, Z -3.0000, A 0.000, B 0.000, C 0.000 }
gfCNCPoint2[11608] = {X 32.2263, Y 8.2450, Z -3.0000, A 0.000, B 0.000, C 0.000 }
gfCNCPoint2[11609] = {X 33.1531, Y 9.4582, Z -3.0000, A 0.000, B 0.000, C 0.000 }
gfCNCPoint2[11610] = {X 33.9860, Y 10.7377, Z -3.0000, A 0.000, B 0.000, C 0.000 }
gfCNCPoint2[11611] = {X 34.8867, Y 12.4168, Z -3.0000, A 0.000, B 0.000, C 0.000 }
gfCNCPoint2[11612] = {X 35.6258, Y 14.1730, Z -3.0000, A 0.000, B 0.000, C 0.000 }
gfCNCPoint2[11613] = {X 36.2224, Y 16.1411, Z -3.0000, A 0.000, B 0.000, C 0.000 }
gfCNCPoint2[11614] = {X 36.6351, Y 18.1558, Z -3.0000, A 0.000, B 0.000, C 0.000 }
gfCNCPoint2[11615] = {X 36.8602, Y 20.2000, Z -3.0000, A 0.000, B 0.000, C 0.000 }
gfCNCPoint2[11616] = {X 36.8961, Y 22.2563, Z -3.0000, A 0.000, B 0.000, C 0.000 }
gfCNCPoint2[11617] = {X 36.7422, Y 24.3070, Z -3.0000, A 0.000, B 0.000, C 0.000 }
gfCNCPoint2[11618] = {X 36.5494, Y 25.5830, Z -3.0000, A 0.000, B 0.000, C 0.000 }
gfCNCPoint2[11619] = {X 36.2830, Y 26.8457, Z -3.0000, A 0.000, B 0.000, C 0.000 }
gfCNCPoint2[11620] = {X 35.8742, Y 28.3053, Z -3.0000, A 0.000, B 0.000, C 0.000 }
gfCNCPoint2[11621] = {X 35.3502, Y 29.7276, Z -3.0000, A 0.000, B 0.000, C 0.000 }
gfCNCPoint2[11622] = {X 34.7143, Y 31.1035, Z -3.0000, A 0.000, B 0.000, C 0.000 }
gfCNCPoint2[11623] = {X 37.2848, Y 36.4136, Z -3.0000, A 0.000, B 0.000, C 0.000 }
gfCNCPoint2[11624] = {X 41.3737, Y 25.4344, Z -3.0000, A 0.000, B 0.000, C 0.000 }
gfCNCPoint2[11625] = {X 45.0743, Y 15.4982, Z -3.0000, A 0.000, B 0.000, C 0.000 }
gfCNCPoint2[11626] = {X 44.7426, Y 14.2853, Z -3.0000, A 0.000, B 0.000, C 0.000 }
gfCNCPoint2[11627] = {X 44.6244, Y 13.0334, Z -3.0000, A 0.000, B 0.000, C 0.000 }
gfCNCPoint2[11628] = {X 44.6242, Y 12.1868, Z -3.0000, A 0.000, B 0.000, C 0.000 }
gfCNCPoint2[11629] = {X 44.6958, Y 11.1684, Z -3.0000, A 0.000, B 0.000, C 0.000 }
gfCNCPoint2[11630] = {X 44.9092, Y 10.1699, Z -3.0000, A 0.000, B 0.000, C 0.000 }
gfCNCPoint2[11631] = {X 45.3323, Y 9.0551, Z -3.0000, A 0.000, B 0.000, C 0.000 }
gfCNCPoint2[11632] = {X 45.9317, Y 8.0242, Z -3.0000, A 0.000, B 0.000, C 0.000 }
gfCNCPoint2[11633] = {X 46.6914, Y 7.1050, Z -3.0000, A 0.000, B 0.000, C 0.000 }
gfCNCPoint2[11634] = {X 42.6031, Y 7.1050, Z -3.0000, A 0.000, B 0.000, C 0.000 }
gfCNCPoint2[11635] = {X 42.6031, Y 4.7050, Z -3.0000, A 0.000, B 0.000, C 0.000 }
gfCNCPoint2[11636] = {X 23.8337, Y 4.7050, Z -3.0000, A 0.000, B 0.000, C 0.000 }
gfCNCPoint2[11637] = {X 25.7628, Y 5.7853, Z -3.0000, A 0.000, B 0.000, C 0.000 }
gfCNCPoint2[11638] = {X 27.5757, Y 7.0510, Z -3.0000, A 0.000, B 0.000, C 0.000 }
gfCNCPoint2[11639] = {X 28.5587, Y 7.8752, Z -3.0000, A 0.000, B 0.000, C 0.000 }
gfCNCPoint2[11640] = {X 29.4801, Y 8.7678, Z -3.0000, A 0.000, B 0.000, C 0.000 }
gfCNCPoint2[11641] = {X 30.6884, Y 10.1631, Z -3.0000, A 0.000, B 0.000, C 0.000 }
gfCNCPoint2[11642] = {X 31.7465, Y 11.6757, Z -3.0000, A 0.000, B 0.000, C 0.000 }
gfCNCPoint2[11643] = {X 32.6428, Y 13.2893, Z -3.0000, A 0.000, B 0.000, C 0.000 }
gfCNCPoint2[11644] = {X 33.3680, Y 14.9868, Z -3.0000, A 0.000, B 0.000, C 0.000 }
gfCNCPoint2[11645] = {X 33.9178, Y 16.8176, Z -3.0000, A 0.000, B 0.000, C 0.000 }
gfCNCPoint2[11646] = {X 34.2892, Y 18.6926, Z -3.0000, A 0.000, B 0.000, C 0.000 }
gfCNCPoint2[11647] = {X 34.4790, Y 20.5947, Z -3.0000, A 0.000, B 0.000, C 0.000 }
gfCNCPoint2[11648] = {X 34.4853, Y 22.5062, Z -3.0000, A 0.000, B 0.000, C 0.000 }
gfCNCPoint2[11649] = {X 34.3081, Y 24.4095, Z -3.0000, A 0.000, B 0.000, C 0.000 }
gfCNCPoint2[11650] = {X 33.9490, Y 26.2870, Z -3.0000, A 0.000, B 0.000, C 0.000 }
gfCNCPoint2[11651] = {X 33.4654, Y 27.9388, Z -3.0000, A 0.000, B 0.000, C 0.000 }
gfCNCPoint2[11652] = {X 32.8131, Y 29.5315, Z -3.0000, A 0.000, B 0.000, C 0.000 }
gfCNCPoint2[11653] = {X 31.9990, Y 31.0479, Z -3.0000, A 0.000, B 0.000, C 0.000 }
gfCNCPoint2[11654] = {X 32.1285, Y 31.2837, Z -3.0000, A 0.000, B 0.000, C 0.000 }
gfCNCPoint2[11655] = {X 32.2510, Y 31.5232, Z -3.0000, A 0.000, B 0.000, C 0.000 }
gfCNCPoint2[11656] = {X 35.3025, Y 37.8269, Z -3.0000, A 0.000, B 0.000, C 0.000 }
gfCNCPoint2[11657] = {X 35.7263, Y 38.8573, Z -3.0000, A 0.000, B 0.000, C 0.000 }
gfCNCPoint2[11658] = {X 36.0224, Y 39.9313, Z -3.0000, A 0.000, B 0.000, C 0.000 }
gfCNCPoint2[11659] = {X 36.1865, Y 41.0332, Z -3.0000, A 0.000, B 0.000, C 0.000 }
gfCNCPoint2[11660] = {X 36.2163, Y 42.1469, Z -3.0000, A 0.000, B 0.000, C 0.000 }
gfCNCPoint2[11661] = {X 36.6305, Y 41.4260, Z -3.0000, A 0.000, B 0.000, C 0.000 }
gfCNCPoint2[11662] = {X 37.1611, Y 40.7858, Z -3.0000, A 0.000, B 0.000, C 0.000 }
gfCNCPoint2[11663] = {X 37.7927, Y 40.2451, Z -3.0000, A 0.000, B 0.000, C 0.000 }
gfCNCPoint2[11664] = {X 38.5069, Y 39.8193, Z -3.0000, A 0.000, B 0.000, C 0.000 }
gfCNCPoint2[11665] = {X 39.0454, Y 38.5337, Z -3.0000, A 0.000, B 0.000, C 0.000 }
gfCNCPoint2[11666] = {X 39.5412, Y 37.2312, Z -3.0000, A 0.000, B 0.000, C 0.000 }
gfCNCPoint2[11667] = {X 47.6703, Y 15.4045, Z -3.0000, A 0.000, B 0.000, C 0.000 }
gfCNCPoint2[11668] = {X 47.3200, Y 14.6512, Z -3.0000, A 0.000, B 0.000, C 0.000 }
gfCNCPoint2[11669] = {X 47.1026, Y 13.8493, Z -3.0000, A 0.000, B 0.000, C 0.000 }
gfCNCPoint2[11670] = {X 47.0244, Y 13.0222, Z -3.0000, A 0.000, B 0.000, C 0.000 }
gfCNCPoint2[11671] = {X 47.0242, Y 12.1868, Z -3.0000, A 0.000, B 0.000, C 0.000 }
gfCNCPoint2[11672] = {X 47.1150, Y 11.2500, Z -3.0000, A 0.000, B 0.000, C 0.000 }
gfCNCPoint2[11673] = {X 47.3839, Y 10.3481, Z -3.0000, A 0.000, B 0.000, C 0.000 }
gfCNCPoint2[11674] = {X 47.8209, Y 9.5145, Z -3.0000, A 0.000, B 0.000, C 0.000 }
gfCNCPoint2[11675] = {X 48.4099, Y 8.7804, Z -3.0000, A 0.000, B 0.000, C 0.000 }
gfCNCPoint2[11676] = {X 49.1544, Y 8.1553, Z -3.0000, A 0.000, B 0.000, C 0.000 }
gfCNCPoint2[11677] = {X 50.0081, Y 7.6903, Z -3.0000, A 0.000, B 0.000, C 0.000 }
gfCNCPoint2[11678] = {X 50.9370, Y 7.4036, Z -3.0000, A 0.000, B 0.000, C 0.000 }
gfCNCPoint2[11679] = {X 51.9042, Y 7.3068, Z -3.0000, A 0.000, B 0.000, C 0.000 }
gfCNCPoint2[11680] = {X 59.6221, Y 7.3068, Z -3.0000, A 0.000, B 0.000, C 0.000 }
gfCNCPoint2[11681] = {X 60.5894, Y 7.4036, Z -3.0000, A 0.000, B 0.000, C 0.000 }
gfCNCPoint2[11682] = {X 61.5183, Y 7.6903, Z -3.0000, A 0.000, B 0.000, C 0.000 }
gfCNCPoint2[11683] = {X 62.3719, Y 8.1553, Z -3.0000, A 0.000, B 0.000, C 0.000 }
gfCNCPoint2[11684] = {X 63.1165, Y 8.7804, Z -3.0000, A 0.000, B 0.000, C 0.000 }
gfCNCPoint2[11685] = {X 63.7054, Y 9.5145, Z -3.0000, A 0.000, B 0.000, C 0.000 }
gfCNCPoint2[11686] = {X 64.1425, Y 10.3481, Z -3.0000, A 0.000, B 0.000, C 0.000 }
gfCNCPoint2[11687] = {X 64.4114, Y 11.2500, Z -3.0000, A 0.000, B 0.000, C 0.000 }
gfCNCPoint2[11688] = {X 64.5021, Y 12.1868, Z -3.0000, A 0.000, B 0.000, C 0.000 }
gfCNCPoint2[11689] = {X 64.5019, Y 13.0237, Z -3.0000, A 0.000, B 0.000, C 0.000 }
gfCNCPoint2[11690] = {X 64.4203, Y 13.8676, Z -3.0000, A 0.000, B 0.000, C 0.000 }
gfCNCPoint2[11691] = {X 64.1940, Y 14.6847, Z -3.0000, A 0.000, B 0.000, C 0.000 }
gfCNCPoint2[11692] = {X 63.8296, Y 15.4502, Z -3.0000, A 0.000, B 0.000, C 0.000 }
gfCNCPoint2[11693] = {X 72.9536, Y 39.8575, Z -3.0000, A 0.000, B 0.000, C 0.000 }
gfCNCPoint2[11694] = {X 73.8438, Y 40.4394, Z -3.0000, A 0.000, B 0.000, C 0.000 }
gfCNCPoint2[11695] = {X 74.5868, Y 41.2003, Z -3.0000, A 0.000, B 0.000, C 0.000 }
gfCNCPoint2[11696] = {X 75.1473, Y 42.1042, Z -3.0000, A 0.000, B 0.000, C 0.000 }
gfCNCPoint2[11697] = {X 75.4987, Y 43.1080, Z -3.0000, A 0.000, B 0.000, C 0.000 }
gfCNCPoint2[11698] = {X 75.6243, Y 44.1640, Z -3.0000, A 0.000, B 0.000, C 0.000 }
gfCNCPoint2[11699] = {X 75.6245, Y 45.0000, Z -3.0000, A 0.000, B 0.000, C 0.000 }
gfCNCPoint2[11700] = {X 75.5307, Y 45.9520, Z -3.0000, A 0.000, B 0.000, C 0.000 }
gfCNCPoint2[11701] = {X 75.2530, Y 46.8675, Z -3.0000, A 0.000, B 0.000, C 0.000 }
gfCNCPoint2[11702] = {X 74.8020, Y 47.7112, Z -3.0000, A 0.000, B 0.000, C 0.000 }
gfCNCPoint2[11703] = {X 74.1951, Y 48.4507, Z -3.0000, A 0.000, B 0.000, C 0.000 }
gfCNCPoint2[11704] = {X 73.4556, Y 49.0576, Z -3.0000, A 0.000, B 0.000, C 0.000 }
gfCNCPoint2[11705] = {X 72.6120, Y 49.5085, Z -3.0000, A 0.000, B 0.000, C 0.000 }
gfCNCPoint2[11706] = {X 71.6965, Y 49.7862, Z -3.0000, A 0.000, B 0.000, C 0.000 }
gfCNCPoint2[11707] = {X 70.7445, Y 49.8800, Z -3.0000, A 0.000, B 0.000, C 0.000 }
gfCNCPoint2[11708] = {X 64.1851, Y 49.8800, Z -3.0000, A 0.000, B 0.000, C 0.000 }
gfCNCPoint2[11709] = {X 63.2331, Y 49.7862, Z -3.0000, A 0.000, B 0.000, C 0.000 }
gfCNCPoint2[11710] = {X 62.3176, Y 49.5085, Z -3.0000, A 0.000, B 0.000, C 0.000 }
gfCNCPoint2[11711] = {X 61.4740, Y 49.0576, Z -3.0000, A 0.000, B 0.000, C 0.000 }
gfCNCPoint2[11712] = {X 60.7345, Y 48.4507, Z -3.0000, A 0.000, B 0.000, C 0.000 }
gfCNCPoint2[11713] = {X 60.1276, Y 47.7112, Z -3.0000, A 0.000, B 0.000, C 0.000 }
gfCNCPoint2[11714] = {X 59.6766, Y 46.8675, Z -3.0000, A 0.000, B 0.000, C 0.000 }
gfCNCPoint2[11715] = {X 59.3989, Y 45.9520, Z -3.0000, A 0.000, B 0.000, C 0.000 }
gfCNCPoint2[11716] = {X 59.3051, Y 45.0000, Z -3.0000, A 0.000, B 0.000, C 0.000 }
gfCNCPoint2[11717] = {X 59.3052, Y 44.2029, Z -3.0000, A 0.000, B 0.000, C 0.000 }
gfCNCPoint2[11718] = {X 59.3848, Y 43.3309, Z -3.0000, A 0.000, B 0.000, C 0.000 }
gfCNCPoint2[11719] = {X 59.6189, Y 42.4872, Z -3.0000, A 0.000, B 0.000, C 0.000 }
gfCNCPoint2[11720] = {X 60.0001, Y 41.6989, Z -3.0000, A 0.000, B 0.000, C 0.000 }
gfCNCPoint2[11721] = {X 59.6159, Y 40.6492, Z -3.0000, A 0.000, B 0.000, C 0.000 }
gfCNCPoint2[11722] = {X 52.4658, Y 40.6492, Z -3.0000, A 0.000, B 0.000, C 0.000 }
gfCNCPoint2[11723] = {X 51.9466, Y 42.0441, Z -3.0000, A 0.000, B 0.000, C 0.000 }
gfCNCPoint2[11724] = {X 52.2215, Y 42.7237, Z -3.0000, A 0.000, B 0.000, C 0.000 }
gfCNCPoint2[11725] = {X 52.3915, Y 43.4367, Z -3.0000, A 0.000, B 0.000, C 0.000 }
gfCNCPoint2[11726] = {X 52.4528, Y 44.1672, Z -3.0000, A 0.000, B 0.000, C 0.000 }
gfCNCPoint2[11727] = {X 52.4529, Y 45.0000, Z -3.0000, A 0.000, B 0.000, C 0.000 }
gfCNCPoint2[11728] = {X 52.3592, Y 45.9520, Z -3.0000, A 0.000, B 0.000, C 0.000 }
gfCNCPoint2[11729] = {X 52.0815, Y 46.8675, Z -3.0000, A 0.000, B 0.000, C 0.000 }
gfCNCPoint2[11730] = {X 51.6305, Y 47.7112, Z -3.0000, A 0.000, B 0.000, C 0.000 }
gfCNCPoint2[11731] = {X 51.0236, Y 48.4507, Z -3.0000, A 0.000, B 0.000, C 0.000 }
gfCNCPoint2[11732] = {X 50.2841, Y 49.0576, Z -3.0000, A 0.000, B 0.000, C 0.000 }
gfCNCPoint2[11733] = {X 49.4404, Y 49.5085, Z -3.0000, A 0.000, B 0.000, C 0.000 }
gfCNCPoint2[11734] = {X 48.5250, Y 49.7862, Z -3.0000, A 0.000, B 0.000, C 0.000 }
gfCNCPoint2[11735] = {X 47.5729, Y 49.8800, Z -3.0000, A 0.000, B 0.000, C 0.000 }
gfCNCPoint2[11736] = {X 40.6393, Y 49.8800, Z -3.0000, A 0.000, B 0.000, C 0.000 }
gfCNCPoint2[11737] = {X 39.6433, Y 49.7773, Z -3.0000, A 0.000, B 0.000, C 0.000 }
gfCNCPoint2[11738] = {X 38.6892, Y 49.4734, Z -3.0000, A 0.000, B 0.000, C 0.000 }
gfCNCPoint2[11739] = {X 37.8173, Y 48.9813, Z -3.0000, A 0.000, B 0.000, C 0.000 }
gfCNCPoint2[11740] = {X 37.0641, Y 48.3215, Z -3.0000, A 0.000, B 0.000, C 0.000 }
gfCNCPoint2[11741] = {X 36.5085, Y 47.5983, Z -3.0000, A 0.000, B 0.000, C 0.000 }
gfCNCPoint2[11742] = {X 36.0972, Y 46.7843, Z -3.0000, A 0.000, B 0.000, C 0.000 }
gfCNCPoint2[11743] = {X 35.8445, Y 45.9080, Z -3.0000, A 0.000, B 0.000, C 0.000 }
gfCNCPoint2[11744] = {X 35.7593, Y 45.0000, Z -3.0000, A 0.000, B 0.000, C 0.000 }
gfCNCPoint2[11745] = {X 35.7593, Y 44.7148, Z -3.0000, A 0.000, B 0.000, C 0.000 }
gfCNCPoint2[11746] = {X 36.2393, Y 44.7148, Z -3.0000, A 0.000, B 0.000, C 0.000 }
gfCNCPoint2[11747] = {X 36.2397, Y 44.1483, Z -3.0000, A 0.000, B 0.000, C 0.000 }
gfCNCPoint2[11748] = {X 36.3681, Y 43.1520, Z -3.0000, A 0.000, B 0.000, C 0.000 }
gfCNCPoint2[11749] = {X 36.7191, Y 42.2108, Z -3.0000, A 0.000, B 0.000, C 0.000 }
gfCNCPoint2[11750] = {X 37.2744, Y 41.3738, Z -3.0000, A 0.000, B 0.000, C 0.000 }
gfCNCPoint2[11751] = {X 38.0050, Y 40.6845, Z -3.0000, A 0.000, B 0.000, C 0.000 }
gfCNCPoint2[11752] = {X 38.8730, Y 40.1789, Z -3.0000, A 0.000, B 0.000, C 0.000 }
gfCNCPoint2[11753] = {X 39.4563, Y 38.7985, Z -3.0000, A 0.000, B 0.000, C 0.000 }
gfCNCPoint2[11754] = {X 39.9911, Y 37.3987, Z -3.0000, A 0.000, B 0.000, C 0.000 }
gfCNCPoint2[11755] = {X 48.2011, Y 15.3544, Z -3.0000, A 0.000, B 0.000, C 0.000 }
gfCNCPoint2[11756] = {X 47.8187, Y 14.6115, Z -3.0000, A 0.000, B 0.000, C 0.000 }
gfCNCPoint2[11757] = {X 47.5835, Y 13.8097, Z -3.0000, A 0.000, B 0.000, C 0.000 }
gfCNCPoint2[11758] = {X 47.5042, Y 12.9779, Z -3.0000, A 0.000, B 0.000, C 0.000 }
gfCNCPoint2[11759] = {X 47.5042, Y 12.1868, Z -3.0000, A 0.000, B 0.000, C 0.000 }
gfCNCPoint2[11760] = {X 47.6145, Y 11.2077, Z -3.0000, A 0.000, B 0.000, C 0.000 }
gfCNCPoint2[11761] = {X 47.9400, Y 10.2777, Z -3.0000, A 0.000, B 0.000, C 0.000 }
gfCNCPoint2[11762] = {X 48.4642, Y 9.4435, Z -3.0000, A 0.000, B 0.000, C 0.000 }
gfCNCPoint2[11763] = {X 49.1609, Y 8.7468, Z -3.0000, A 0.000, B 0.000, C 0.000 }
gfCNCPoint2[11764] = {X 49.9951, Y 8.2226, Z -3.0000, A 0.000, B 0.000, C 0.000 }
gfCNCPoint2[11765] = {X 50.9251, Y 7.8971, Z -3.0000, A 0.000, B 0.000, C 0.000 }
gfCNCPoint2[11766] = {X 51.9042, Y 7.7868, Z -3.0000, A 0.000, B 0.000, C 0.000 }
gfCNCPoint2[11767] = {X 59.6221, Y 7.7868, Z -3.0000, A 0.000, B 0.000, C 0.000 }
gfCNCPoint2[11768] = {X 60.6012, Y 7.8971, Z -3.0000, A 0.000, B 0.000, C 0.000 }
gfCNCPoint2[11769] = {X 61.5312, Y 8.2226, Z -3.0000, A 0.000, B 0.000, C 0.000 }
gfCNCPoint2[11770] = {X 62.3655, Y 8.7468, Z -3.0000, A 0.000, B 0.000, C 0.000 }
gfCNCPoint2[11771] = {X 63.0622, Y 9.4435, Z -3.0000, A 0.000, B 0.000, C 0.000 }
gfCNCPoint2[11772] = {X 63.5864, Y 10.2777, Z -3.0000, A 0.000, B 0.000, C 0.000 }
gfCNCPoint2[11773] = {X 63.9118, Y 11.2077, Z -3.0000, A 0.000, B 0.000, C 0.000 }
gfCNCPoint2[11774] = {X 64.0221, Y 12.1868, Z -3.0000, A 0.000, B 0.000, C 0.000 }
gfCNCPoint2[11775] = {X 64.0219, Y 13.0233, Z -3.0000, A 0.000, B 0.000, C 0.000 }
gfCNCPoint2[11776] = {X 63.9335, Y 13.8565, Z -3.0000, A 0.000, B 0.000, C 0.000 }
gfCNCPoint2[11777] = {X 63.6888, Y 14.6579, Z -3.0000, A 0.000, B 0.000, C 0.000 }
gfCNCPoint2[11778] = {X 63.2966, Y 15.3984, Z -3.0000, A 0.000, B 0.000, C 0.000 }
gfCNCPoint2[11779] = {X 63.5001, Y 15.9354, Z -3.0000, A 0.000, B 0.000, C 0.000 }
gfCNCPoint2[11780] = {X 66.1097, Y 22.8602, Z -3.0000, A 0.000, B 0.000, C 0.000 }
gfCNCPoint2[11781] = {X 72.2837, Y 39.4716, Z -3.0000, A 0.000, B 0.000, C 0.000 }
gfCNCPoint2[11782] = {X 72.5766, Y 40.2084, Z -3.0000, A 0.000, B 0.000, C 0.000 }
gfCNCPoint2[11783] = {X 73.4343, Y 40.7267, Z -3.0000, A 0.000, B 0.000, C 0.000 }
gfCNCPoint2[11784] = {X 74.1525, Y 41.4258, Z -3.0000, A 0.000, B 0.000, C 0.000 }
gfCNCPoint2[11785] = {X 74.6939, Y 42.2692, Z -3.0000, A 0.000, B 0.000, C 0.000 }
gfCNCPoint2[11786] = {X 75.0303, Y 43.2132, Z -3.0000, A 0.000, B 0.000, C 0.000 }
gfCNCPoint2[11787] = {X 75.1445, Y 44.2089, Z -3.0000, A 0.000, B 0.000, C 0.000 }
gfCNCPoint2[11788] = {X 75.1445, Y 45.0000, Z -3.0000, A 0.000, B 0.000, C 0.000 }
gfCNCPoint2[11789] = {X 75.0341, Y 45.9791, Z -3.0000, A 0.000, B 0.000, C 0.000 }
gfCNCPoint2[11790] = {X 74.7087, Y 46.9091, Z -3.0000, A 0.000, B 0.000, C 0.000 }
gfCNCPoint2[11791] = {X 74.1845, Y 47.7434, Z -3.0000, A 0.000, B 0.000, C 0.000 }
gfCNCPoint2[11792] = {X 73.4878, Y 48.4401, Z -3.0000, A 0.000, B 0.000, C 0.000 }
gfCNCPoint2[11793] = {X 72.6535, Y 48.9643, Z -3.0000, A 0.000, B 0.000, C 0.000 }
gfCNCPoint2[11794] = {X 71.7236, Y 49.2897, Z -3.0000, A 0.000, B 0.000, C 0.000 }
gfCNCPoint2[11795] = {X 70.7445, Y 49.4000, Z -3.0000, A 0.000, B 0.000, C 0.000 }
gfCNCPoint2[11796] = {X 64.1851, Y 49.4000, Z -3.0000, A 0.000, B 0.000, C 0.000 }
gfCNCPoint2[11797] = {X 63.2060, Y 49.2897, Z -3.0000, A 0.000, B 0.000, C 0.000 }
gfCNCPoint2[11798] = {X 62.2760, Y 48.9643, Z -3.0000, A 0.000, B 0.000, C 0.000 }
gfCNCPoint2[11799] = {X 61.4418, Y 48.4401, Z -3.0000, A 0.000, B 0.000, C 0.000 }
gfCNCPoint2[11800] = {X 60.7451, Y 47.7434, Z -3.0000, A 0.000, B 0.000, C 0.000 }
gfCNCPoint2[11801] = {X 60.2209, Y 46.9091, Z -3.0000, A 0.000, B 0.000, C 0.000 }
gfCNCPoint2[11802] = {X 59.8955, Y 45.9791, Z -3.0000, A 0.000, B 0.000, C 0.000 }
gfCNCPoint2[11803] = {X 59.7851, Y 45.0000, Z -3.0000, A 0.000, B 0.000, C 0.000 }
gfCNCPoint2[11804] = {X 59.7856, Y 44.1483, Z -3.0000, A 0.000, B 0.000, C 0.000 }
gfCNCPoint2[11805] = {X 59.8784, Y 43.3076, Z -3.0000, A 0.000, B 0.000, C 0.000 }
gfCNCPoint2[11806] = {X 60.1304, Y 42.5003, Z -3.0000, A 0.000, B 0.000, C 0.000 }
gfCNCPoint2[11807] = {X 60.5322, Y 41.7561, Z -3.0000, A 0.000, B 0.000, C 0.000 }
gfCNCPoint2[11808] = {X 59.9513, Y 40.1692, Z -3.0000, A 0.000, B 0.000, C 0.000 }
gfCNCPoint2[11809] = {X 52.1323, Y 40.1692, Z -3.0000, A 0.000, B 0.000, C 0.000 }
gfCNCPoint2[11810] = {X 51.4221, Y 42.0772, Z -3.0000, A 0.000, B 0.000, C 0.000 }
gfCNCPoint2[11811] = {X 51.7252, Y 42.7532, Z -3.0000, A 0.000, B 0.000, C 0.000 }
gfCNCPoint2[11812] = {X 51.9106, Y 43.4706, Z -3.0000, A 0.000, B 0.000, C 0.000 }
gfCNCPoint2[11813] = {X 51.9729, Y 44.2089, Z -3.0000, A 0.000, B 0.000, C 0.000 }
gfCNCPoint2[11814] = {X 51.9729, Y 45.0000, Z -3.0000, A 0.000, B 0.000, C 0.000 }
gfCNCPoint2[11815] = {X 51.8626, Y 45.9791, Z -3.0000, A 0.000, B 0.000, C 0.000 }
gfCNCPoint2[11816] = {X 51.5372, Y 46.9091, Z -3.0000, A 0.000, B 0.000, C 0.000 }
gfCNCPoint2[11817] = {X 51.0130, Y 47.7434, Z -3.0000, A 0.000, B 0.000, C 0.000 }
gfCNCPoint2[11818] = {X 50.3163, Y 48.4401, Z -3.0000, A 0.000, B 0.000, C 0.000 }
gfCNCPoint2[11819] = {X 49.4820, Y 48.9643, Z -3.0000, A 0.000, B 0.000, C 0.000 }
gfCNCPoint2[11820] = {X 48.5520, Y 49.2897, Z -3.0000, A 0.000, B 0.000, C 0.000 }
gfCNCPoint2[11821] = {X 47.5729, Y 49.4000, Z -3.0000, A 0.000, B 0.000, C 0.000 }
gfCNCPoint2[11822] = {X 40.6393, Y 49.4000, Z -3.0000, A 0.000, B 0.000, C 0.000 }
gfCNCPoint2[11823] = {X 39.6602, Y 49.2897, Z -3.0000, A 0.000, B 0.000, C 0.000 }
gfCNCPoint2[11824] = {X 38.7302, Y 48.9643, Z -3.0000, A 0.000, B 0.000, C 0.000 }
gfCNCPoint2[11825] = {X 37.8959, Y 48.4401, Z -3.0000, A 0.000, B 0.000, C 0.000 }
gfCNCPoint2[11826] = {X 37.1992, Y 47.7434, Z -3.0000, A 0.000, B 0.000, C 0.000 }
gfCNCPoint2[11827] = {X 36.6750, Y 46.9091, Z -3.0000, A 0.000, B 0.000, C 0.000 }
gfCNCPoint2[11828] = {X 36.3496, Y 45.9791, Z -3.0000, A 0.000, B 0.000, C 0.000 }
gfCNCPoint2[11829] = {X 36.2393, Y 45.0000, Z -3.0000, A 0.000, B 0.000, C 0.000 }
gfCNCPoint2[11830] = {X 36.2393, Y 44.7148, Z -3.0000, A 0.000, B 0.000, C 0.000 }
gfCNCPoint2[11831] = {X 35.7593, Y 44.7148, Z -3.0000, A 0.000, B 0.000, C 0.000 }
gfCNCPoint2[11832] = {X 35.2211, Y 46.0074, Z -3.0000, A 0.000, B 0.000, C 0.000 }
gfCNCPoint2[11833] = {X 34.4930, Y 47.2034, Z -3.0000, A 0.000, B 0.000, C 0.000 }
gfCNCPoint2[11834] = {X 33.5918, Y 48.2750, Z -3.0000, A 0.000, B 0.000, C 0.000 }
gfCNCPoint2[11835] = {X 33.2092, Y 48.6435, Z -3.0000, A 0.000, B 0.000, C 0.000 }
gfCNCPoint2[11836] = {X 32.8060, Y 48.9892, Z -3.0000, A 0.000, B 0.000, C 0.000 }
gfCNCPoint2[11837] = {X 32.2657, Y 49.4260, Z -3.0000, A 0.000, B 0.000, C 0.000 }
gfCNCPoint2[11838] = {X 31.1802, Y 50.1801, Z -3.0000, A 0.000, B 0.000, C 0.000 }
gfCNCPoint2[11839] = {X 29.9980, Y 50.7711, Z -3.0000, A 0.000, B 0.000, C 0.000 }
gfCNCPoint2[11840] = {X 28.7434, Y 51.1870, Z -3.0000, A 0.000, B 0.000, C 0.000 }
gfCNCPoint2[11841] = {X 27.4422, Y 51.4191, Z -3.0000, A 0.000, B 0.000, C 0.000 }
gfCNCPoint2[11842] = {X 26.1212, Y 51.4627, Z -3.0000, A 0.000, B 0.000, C 0.000 }
gfCNCPoint2[11843] = {X 24.0665, Y 52.4198, Z -3.0000, A 0.000, B 0.000, C 0.000 }
gfCNCPoint2[11844] = {X 21.9507, Y 53.2329, Z -3.0000, A 0.000, B 0.000, C 0.000 }
gfCNCPoint2[11845] = {X 19.6217, Y 53.9647, Z -3.0000, A 0.000, B 0.000, C 0.000 }
gfCNCPoint2[11846] = {X 17.2373, Y 54.4886, Z -3.0000, A 0.000, B 0.000, C 0.000 }
gfCNCPoint2[11847] = {X 14.8160, Y 54.8005, Z -3.0000, A 0.000, B 0.000, C 0.000 }
gfCNCPoint2[11848] = {X 12.3767, Y 54.8980, Z -3.0000, A 0.000, B 0.000, C 0.000 }
gfCNCPoint2[11849] = {X 9.9383, Y 54.7803, Z -3.0000, A 0.000, B 0.000, C 0.000 }
gfCNCPoint2[11850] = {X 7.5197, Y 54.4484, Z -3.0000, A 0.000, B 0.000, C 0.000 }
gfCNCPoint2[11851] = {X 6.1002, Y 54.1499, Z -3.0000, A 0.000, B 0.000, C 0.000 }
gfCNCPoint2[11852] = {X 4.7035, Y 53.7586, Z -3.0000, A 0.000, B 0.000, C 0.000 }
gfCNCPoint2[11853] = {X 4.7035, Y 95.2950, Z -3.0000, A 0.000, B 0.000, C 0.000 }
gfCNCPoint2[11854] = {X 117.9387, Y 95.2950, Z -3.0000, A 0.000, B 0.000, C 0.000 }
gfCNCPoint2[11855] = {X 118.3616, Y 94.0776, Z -3.0000, A 0.000, B 0.000, C 0.000 }
gfCNCPoint2[11856] = {X 118.9925, Y 92.9539, Z -3.0000, A 0.000, B 0.000, C 0.000 }
gfCNCPoint2[11857] = {X 119.8117, Y 91.9591, Z -3.0000, A 0.000, B 0.000, C 0.000 }
gfCNCPoint2[11858] = {X 120.7934, Y 91.1243, Z -3.0000, A 0.000, B 0.000, C 0.000 }
gfCNCPoint2[11859] = {X 121.9070, Y 90.4757, Z -3.0000, A 0.000, B 0.000, C 0.000 }
gfCNCPoint2[11860] = {X 123.1174, Y 90.0336, Z -3.0000, A 0.000, B 0.000, C 0.000 }
gfCNCPoint2[11861] = {X 124.3869, Y 89.8118, Z -3.0000, A 0.000, B 0.000, C 0.000 }
gfCNCPoint2[11862] = {X 125.0466, Y 89.7124, Z -3.0000, A 0.000, B 0.000, C 0.000 }
gfCNCPoint2[11863] = {X 125.3569, Y 89.6657, Z -3.0000, A 0.000, B 0.000, C 0.000 }
gfCNCPoint2[11864] = {X 125.6655, Y 89.6088, Z -3.0000, A 0.000, B 0.000, C 0.000 }
gfCNCPoint2[11865] = {X 126.4923, Y 88.7982, Z -3.0000, A 0.000, B 0.000, C 0.000 }
gfCNCPoint2[11866] = {X 127.2849, Y 87.9541, Z -3.0000, A 0.000, B 0.000, C 0.000 }
gfCNCPoint2[11867] = {X 152.2077, Y 60.5853, Z -3.0000, A 0.000, B 0.000, C 0.000 }
gfCNCPoint2[11868] = {X 152.0685, Y 59.7902, Z -3.0000, A 0.000, B 0.000, C 0.000 }
gfCNCPoint2[11869] = {X 152.0181, Y 58.9845, Z -3.0000, A 0.000, B 0.000, C 0.000 }
gfCNCPoint2[11870] = {X 152.0180, Y 58.0000, Z -3.0000, A 0.000, B 0.000, C 0.000 }
gfCNCPoint2[11871] = {X 152.1286, Y 56.7358, Z -3.0000, A 0.000, B 0.000, C 0.000 }
gfCNCPoint2[11872] = {X 152.4570, Y 55.5101, Z -3.0000, A 0.000, B 0.000, C 0.000 }
gfCNCPoint2[11873] = {X 152.9933, Y 54.3600, Z -3.0000, A 0.000, B 0.000, C 0.000 }
gfCNCPoint2[11874] = {X 153.7212, Y 53.3205, Z -3.0000, A 0.000, B 0.000, C 0.000 }
gfCNCPoint2[11875] = {X 154.6185, Y 52.4232, Z -3.0000, A 0.000, B 0.000, C 0.000 }
gfCNCPoint2[11876] = {X 155.6580, Y 51.6953, Z -3.0000, A 0.000, B 0.000, C 0.000 }
gfCNCPoint2[11877] = {X 156.8081, Y 51.1590, Z -3.0000, A 0.000, B 0.000, C 0.000 }
gfCNCPoint2[11878] = {X 158.0338, Y 50.8306, Z -3.0000, A 0.000, B 0.000, C 0.000 }
gfCNCPoint2[11879] = {X 159.2980, Y 50.7200, Z -3.0000, A 0.000, B 0.000, C 0.000 }
gfCNCPoint2[11880] = {X 178.5335, Y 50.7200, Z -3.0000, A 0.000, B 0.000, C 0.000 }
gfCNCPoint2[11881] = {X 179.7868, Y 50.8287, Z -3.0000, A 0.000, B 0.000, C 0.000 }
gfCNCPoint2[11882] = {X 181.0027, Y 51.1515, Z -3.0000, A 0.000, B 0.000, C 0.000 }
gfCNCPoint2[11883] = {X 182.1449, Y 51.6789, Z -3.0000, A 0.000, B 0.000, C 0.000 }
gfCNCPoint2[11884] = {X 183.1792, Y 52.3950, Z -3.0000, A 0.000, B 0.000, C 0.000 }
gfCNCPoint2[11885] = {X 184.0876, Y 53.2936, Z -3.0000, A 0.000, B 0.000, C 0.000 }
gfCNCPoint2[11886] = {X 184.8249, Y 54.3371, Z -3.0000, A 0.000, B 0.000, C 0.000 }
gfCNCPoint2[11887] = {X 185.3684, Y 55.4936, Z -3.0000, A 0.000, B 0.000, C 0.000 }
gfCNCPoint2[11888] = {X 185.7014, Y 56.7272, Z -3.0000, A 0.000, B 0.000, C 0.000 }
gfCNCPoint2[11889] = {X 185.8135, Y 58.0000, Z -3.0000, A 0.000, B 0.000, C 0.000 }
gfCNCPoint2[11890] = {X 185.8133, Y 58.9942, Z -3.0000, A 0.000, B 0.000, C 0.000 }
gfCNCPoint2[11891] = {X 185.7647, Y 59.7752, Z -3.0000, A 0.000, B 0.000, C 0.000 }
gfCNCPoint2[11892] = {X 185.6327, Y 60.5466, Z -3.0000, A 0.000, B 0.000, C 0.000 }
gfCNCPoint2[11893] = {X 211.6604, Y 88.9544, Z -3.0000, A 0.000, B 0.000, C 0.000 }
gfCNCPoint2[11894] = {X 212.0329, Y 89.3394, Z -3.0000, A 0.000, B 0.000, C 0.000 }
gfCNCPoint2[11895] = {X 212.4256, Y 89.7037, Z -3.0000, A 0.000, B 0.000, C 0.000 }
gfCNCPoint2[11896] = {X 212.6034, Y 89.7418, Z -3.0000, A 0.000, B 0.000, C 0.000 }
gfCNCPoint2[11897] = {X 213.4472, Y 89.8481, Z -3.0000, A 0.000, B 0.000, C 0.000 }
gfCNCPoint2[11898] = {X 214.4295, Y 89.7712, Z -3.0000, A 0.000, B 0.000, C 0.000 }
gfCNCPoint2[11899] = {X 215.4134, Y 89.7175, Z -3.0000, A 0.000, B 0.000, C 0.000 }
gfCNCPoint2[11900] = {X 215.6263, Y 89.6939, Z -3.0000, A 0.000, B 0.000, C 0.000 }
gfCNCPoint2[11901] = {X 215.8220, Y 89.6068, Z -3.0000, A 0.000, B 0.000, C 0.000 }
gfCNCPoint2[11902] = {X 239.3470, Y 74.5356, Z -3.0000, A 0.000, B 0.000, C 0.000 }
gfCNCPoint2[11903] = {X 220.5437, Y 67.1563, Z -3.0000, A 0.000, B 0.000, C 0.000 }
gfCNCPoint2[11904] = {X 219.0952, Y 66.6702, Z -3.0000, A 0.000, B 0.000, C 0.000 }
gfCNCPoint2[11905] = {X 217.6005, Y 66.3533, Z -3.0000, A 0.000, B 0.000, C 0.000 }
gfCNCPoint2[11906] = {X 216.0794, Y 66.2097, Z -3.0000, A 0.000, B 0.000, C 0.000 }
gfCNCPoint2[11907] = {X 214.8527, Y 66.0624, Z -3.0000, A 0.000, B 0.000, C 0.000 }
gfCNCPoint2[11908] = {X 213.6685, Y 65.7098, Z -3.0000, A 0.000, B 0.000, C 0.000 }
gfCNCPoint2[11909] = {X 212.5610, Y 65.1620, Z -3.0000, A 0.000, B 0.000, C 0.000 }
gfCNCPoint2[11910] = {X 211.5621, Y 64.4348, Z -3.0000, A 0.000, B 0.000, C 0.000 }
gfCNCPoint2[11911] = {X 210.7005, Y 63.5491, Z -3.0000, A 0.000, B 0.000, C 0.000 }
gfCNCPoint2[11912] = {X 210.0012, Y 62.5305, Z -3.0000, A 0.000, B 0.000, C 0.000 }
gfCNCPoint2[11913] = {X 209.4842, Y 61.4083, Z -3.0000, A 0.000, B 0.000, C 0.000 }
gfCNCPoint2[11914] = {X 209.1644, Y 60.2148, Z -3.0000, A 0.000, B 0.000, C 0.000 }
gfCNCPoint2[11915] = {X 209.0510, Y 58.9845, Z -3.0000, A 0.000, B 0.000, C 0.000 }
gfCNCPoint2[11916] = {X 209.0508, Y 58.0000, Z -3.0000, A 0.000, B 0.000, C 0.000 }
gfCNCPoint2[11917] = {X 209.1477, Y 56.8162, Z -3.0000, A 0.000, B 0.000, C 0.000 }
gfCNCPoint2[11918] = {X 209.4358, Y 55.6638, Z -3.0000, A 0.000, B 0.000, C 0.000 }
gfCNCPoint2[11919] = {X 209.9075, Y 54.5737, Z -3.0000, A 0.000, B 0.000, C 0.000 }
gfCNCPoint2[11920] = {X 210.5502, Y 53.5748, Z -3.0000, A 0.000, B 0.000, C 0.000 }
gfCNCPoint2[11921] = {X 211.3467, Y 52.6937, Z -3.0000, A 0.000, B 0.000, C 0.000 }
gfCNCPoint2[11922] = {X 212.2759, Y 51.9538, Z -3.0000, A 0.000, B 0.000, C 0.000 }
gfCNCPoint2[11923] = {X 213.3131, Y 51.3749, Z -3.0000, A 0.000, B 0.000, C 0.000 }
gfCNCPoint2[11924] = {X 214.4306, Y 50.9724, Z -3.0000, A 0.000, B 0.000, C 0.000 }
gfCNCPoint2[11925] = {X 215.3724, Y 50.7834, Z -3.0000, A 0.000, B 0.000, C 0.000 }
gfCNCPoint2[11926] = {X 216.3308, Y 50.7200, Z -3.0000, A 0.000, B 0.000, C 0.000 }
gfCNCPoint2[11927] = {X 237.2617, Y 50.7200, Z -3.0000, A 0.000, B 0.000, C 0.000 }
gfCNCPoint2[11928] = {X 238.3057, Y 50.7953, Z -3.0000, A 0.000, B 0.000, C 0.000 }
gfCNCPoint2[11929] = {X 239.3282, Y 51.0195, Z -3.0000, A 0.000, B 0.000, C 0.000 }
gfCNCPoint2[11930] = {X 240.3080, Y 51.3880, Z -3.0000, A 0.000, B 0.000, C 0.000 }
gfCNCPoint2[11931] = {X 241.2247, Y 51.8932, Z -3.0000, A 0.000, B 0.000, C 0.000 }
gfCNCPoint2[11932] = {X 242.0742, Y 52.5375, Z -3.0000, A 0.000, B 0.000, C 0.000 }
gfCNCPoint2[11933] = {X 242.8204, Y 53.2990, Z -3.0000, A 0.000, B 0.000, C 0.000 }
gfCNCPoint2[11934] = {X 243.4474, Y 54.1613, Z -3.0000, A 0.000, B 0.000, C 0.000 }
gfCNCPoint2[11935] = {X 243.9417, Y 55.1059, Z -3.0000, A 0.000, B 0.000, C 0.000 }
gfCNCPoint2[11936] = {X 244.2928, Y 56.1126, Z -3.0000, A 0.000, B 0.000, C 0.000 }
gfCNCPoint2[11937] = {X 248.5775, Y 57.7829, Z -3.0000, A 0.000, B 0.000, C 0.000 }
gfCNCPoint2[11938] = {X 272.6731, Y 67.3436, Z -3.0000, A 0.000, B 0.000, C 0.000 }
gfCNCPoint2[11939] = {X 272.6730, Y 65.2844, Z -3.0000, A 0.000, B 0.000, C 0.000 }
gfCNCPoint2[11940] = {X 271.6656, Y 64.6033, Z -3.0000, A 0.000, B 0.000, C 0.000 }
gfCNCPoint2[11941] = {X 270.7857, Y 63.7640, Z -3.0000, A 0.000, B 0.000, C 0.000 }
gfCNCPoint2[11942] = {X 270.0577, Y 62.7900, Z -3.0000, A 0.000, B 0.000, C 0.000 }
gfCNCPoint2[11943] = {X 269.5020, Y 61.7083, Z -3.0000, A 0.000, B 0.000, C 0.000 }
gfCNCPoint2[11944] = {X 269.2029, Y 60.8264, Z -3.0000, A 0.000, B 0.000, C 0.000 }
gfCNCPoint2[11945] = {X 269.0189, Y 59.9134, Z -3.0000, A 0.000, B 0.000, C 0.000 }
gfCNCPoint2[11946] = {X 268.9529, Y 58.9845, Z -3.0000, A 0.000, B 0.000, C 0.000 }
gfCNCPoint2[11947] = {X 268.9527, Y 58.0000, Z -3.0000, A 0.000, B 0.000, C 0.000 }
gfCNCPoint2[11948] = {X 269.0633, Y 56.7358, Z -3.0000, A 0.000, B 0.000, C 0.000 }
gfCNCPoint2[11949] = {X 269.3917, Y 55.5101, Z -3.0000, A 0.000, B 0.000, C 0.000 }
gfCNCPoint2[11950] = {X 269.9280, Y 54.3600, Z -3.0000, A 0.000, B 0.000, C 0.000 }
gfCNCPoint2[11951] = {X 270.6559, Y 53.3205, Z -3.0000, A 0.000, B 0.000, C 0.000 }
gfCNCPoint2[11952] = {X 271.5532, Y 52.4232, Z -3.0000, A 0.000, B 0.000, C 0.000 }
gfCNCPoint2[11953] = {X 272.5927, Y 51.6953, Z -3.0000, A 0.000, B 0.000, C 0.000 }
gfCNCPoint2[11954] = {X 273.7428, Y 51.1590, Z -3.0000, A 0.000, B 0.000, C 0.000 }
gfCNCPoint2[11955] = {X 274.9685, Y 50.8306, Z -3.0000, A 0.000, B 0.000, C 0.000 }
gfCNCPoint2[11956] = {X 276.2327, Y 50.7200, Z -3.0000, A 0.000, B 0.000, C 0.000 }
gfCNCPoint2[11957] = {X 292.7731, Y 50.7200, Z -3.0000, A 0.000, B 0.000, C 0.000 }
gfCNCPoint2[11958] = {X 293.4209, Y 50.7489, Z -3.0000, A 0.000, B 0.000, C 0.000 }
gfCNCPoint2[11959] = {X 294.0636, Y 50.8353, Z -3.0000, A 0.000, B 0.000, C 0.000 }
gfCNCPoint2[11960] = {X 294.7295, Y 50.9878, Z -3.0000, A 0.000, B 0.000, C 0.000 }
gfCNCPoint2[11961] = {X 295.3782, Y 51.2021, Z -3.0000, A 0.000, B 0.000, C 0.000 }
gfCNCPoint2[11962] = {X 298.3089, Y 43.5548, Z -3.0000, A 0.000, B 0.000, C 0.000 }
gfCNCPoint2[11963] = {X 298.4822, Y 42.5310, Z -3.0000, A 0.000, B 0.000, C 0.000 }
gfCNCPoint2[11964] = {X 298.7928, Y 41.5402, Z -3.0000, A 0.000, B 0.000, C 0.000 }
gfCNCPoint2[11965] = {X 299.2349, Y 40.6007, Z -3.0000, A 0.000, B 0.000, C 0.000 }
gfCNCPoint2[11966] = {X 299.8004, Y 39.7298, Z -3.0000, A 0.000, B 0.000, C 0.000 }
gfCNCPoint2[11967] = {X 299.8004, Y 36.9943, Z -3.0000, A 0.000, B 0.000, C 0.000 }
gfCNCPoint2[11968] = {X 296.8136, Y 36.9943, Z -3.0000, A 0.000, B 0.000, C 0.000 }
gfCNCPoint2[11969] = {X 296.8132, Y 39.7489, Z -3.0000, A 0.000, B 0.000, C 0.000 }
gfCNCPoint2[11970] = {X 297.3847, Y 40.6118, Z -3.0000, A 0.000, B 0.000, C 0.000 }
gfCNCPoint2[11971] = {X 297.8299, Y 41.5462, Z -3.0000, A 0.000, B 0.000, C 0.000 }
gfCNCPoint2[11972] = {X 298.1400, Y 42.5337, Z -3.0000, A 0.000, B 0.000, C 0.000 }
gfCNCPoint2[11973] = {X 298.3089, Y 43.5548, Z -3.0000, A 0.000, B 0.000, C 0.000 }
gfCNCPoint2[11974] = {X 296.2371, Y 48.9610, Z -3.0000, A 0.000, B 0.000, C 0.000 }
gfCNCPoint2[11975] = {X 296.6128, Y 49.1141, Z -3.0000, A 0.000, B 0.000, C 0.000 }
gfCNCPoint2[11976] = {X 296.9817, Y 49.2828, Z -3.0000, A 0.000, B 0.000, C 0.000 }
gfCNCPoint2[11977] = {X 297.2571, Y 49.4212, Z -3.0000, A 0.000, B 0.000, C 0.000 }
gfCNCPoint2[11978] = {X 297.5280, Y 49.5683, Z -3.0000, A 0.000, B 0.000, C 0.000 }
gfCNCPoint2[11979] = {X 298.7174, Y 50.3602, Z -3.0000, A 0.000, B 0.000, C 0.000 }
gfCNCPoint2[11980] = {X 299.7774, Y 51.3185, Z -3.0000, A 0.000, B 0.000, C 0.000 }
gfCNCPoint2[11981] = {X 300.6847, Y 52.4224, Z -3.0000, A 0.000, B 0.000, C 0.000 }
gfCNCPoint2[11982] = {X 301.5914, Y 51.3191, Z -3.0000, A 0.000, B 0.000, C 0.000 }
gfCNCPoint2[11983] = {X 302.6506, Y 50.3611, Z -3.0000, A 0.000, B 0.000, C 0.000 }
gfCNCPoint2[11984] = {X 303.8393, Y 49.5695, Z -3.0000, A 0.000, B 0.000, C 0.000 }
gfCNCPoint2[11985] = {X 302.8989, Y 49.0956, Z -3.0000, A 0.000, B 0.000, C 0.000 }
gfCNCPoint2[11986] = {X 302.0820, Y 48.4310, Z -3.0000, A 0.000, B 0.000, C 0.000 }
gfCNCPoint2[11987] = {X 301.4268, Y 47.6067, Z -3.0000, A 0.000, B 0.000, C 0.000 }
gfCNCPoint2[11988] = {X 300.9636, Y 46.6610, Z -3.0000, A 0.000, B 0.000, C 0.000 }
gfCNCPoint2[11989] = {X 300.7923, Y 46.0759, Z -3.0000, A 0.000, B 0.000, C 0.000 }
gfCNCPoint2[11990] = {X 300.6953, Y 45.4741, Z -3.0000, A 0.000, B 0.000, C 0.000 }
gfCNCPoint2[11991] = {X 300.6790, Y 45.2570, Z -3.0000, A 0.000, B 0.000, C 0.000 }
gfCNCPoint2[11992] = {X 300.6724, Y 45.0393, Z -3.0000, A 0.000, B 0.000, C 0.000 }
gfCNCPoint2[11993] = {X 300.6725, Y 44.1875, Z -3.0000, A 0.000, B 0.000, C 0.000 }
gfCNCPoint2[11994] = {X 300.6810, Y 43.9903, Z -3.0000, A 0.000, B 0.000, C 0.000 }
gfCNCPoint2[11995] = {X 300.6970, Y 43.7936, Z -3.0000, A 0.000, B 0.000, C 0.000 }
gfCNCPoint2[11996] = {X 300.8618, Y 42.9138, Z -3.0000, A 0.000, B 0.000, C 0.000 }
gfCNCPoint2[11997] = {X 301.1741, Y 42.0749, Z -3.0000, A 0.000, B 0.000, C 0.000 }
gfCNCPoint2[11998] = {X 301.6247, Y 41.3015, Z -3.0000, A 0.000, B 0.000, C 0.000 }
gfCNCPoint2[11999] = {X 302.2004, Y 40.6161, Z -3.0000, A 0.000, B 0.000, C 0.000 }
gfCNCPoint2[12000] = {X 302.2004, Y 34.5943, Z -3.0000, A 0.000, B 0.000, C 0.000 }
gfCNCPoint2[12001] = {X 294.4139, Y 34.5943, Z -3.0000, A 0.000, B 0.000, C 0.000 }
gfCNCPoint2[12002] = {X 294.4131, Y 40.6558, Z -3.0000, A 0.000, B 0.000, C 0.000 }
gfCNCPoint2[12003] = {X 294.9936, Y 41.3230, Z -3.0000, A 0.000, B 0.000, C 0.000 }
gfCNCPoint2[12004] = {X 295.4469, Y 42.0823, Z -3.0000, A 0.000, B 0.000, C 0.000 }
gfCNCPoint2[12005] = {X 295.7588, Y 42.9098, Z -3.0000, A 0.000, B 0.000, C 0.000 }
gfCNCPoint2[12006] = {X 295.9194, Y 43.7795, Z -3.0000, A 0.000, B 0.000, C 0.000 }
gfCNCPoint2[12007] = {X 295.9349, Y 43.9940, Z -3.0000, A 0.000, B 0.000, C 0.000 }
gfCNCPoint2[12008] = {X 295.9411, Y 44.2089, Z -3.0000, A 0.000, B 0.000, C 0.000 }
gfCNCPoint2[12009] = {X 295.9411, Y 45.0000, Z -3.0000, A 0.000, B 0.000, C 0.000 }
gfCNCPoint2[12010] = {X 295.9354, Y 45.2373, Z -3.0000, A 0.000, B 0.000, C 0.000 }
gfCNCPoint2[12011] = {X 295.9180, Y 45.4741, Z -3.0000, A 0.000, B 0.000, C 0.000 }
gfCNCPoint2[12012] = {X 298.3067, Y 45.7073, Z -3.0000, A 0.000, B 0.000, C 0.000 }
gfCNCPoint2[12013] = {X 298.2010, Y 46.4214, Z -3.0000, A 0.000, B 0.000, C 0.000 }
gfCNCPoint2[12014] = {X 298.0252, Y 47.1215, Z -3.0000, A 0.000, B 0.000, C 0.000 }
gfCNCPoint2[12015] = {X 298.3689, Y 47.2942, Z -3.0000, A 0.000, B 0.000, C 0.000 }
gfCNCPoint2[12016] = {X 298.7069, Y 47.4778, Z -3.0000, A 0.000, B 0.000, C 0.000 }
gfCNCPoint2[12017] = {X 298.4514, Y 46.6051, Z -3.0000, A 0.000, B 0.000, C 0.000 }
gfCNCPoint2[12018] = {X 298.3067, Y 45.7073, Z -3.0000, A 0.000, B 0.000, C 0.000 }
gfCNCPoint2[12019] = {X 295.9180, Y 45.4741, Z -3.0000, A 0.000, B 0.000, C 0.000 }
gfCNCPoint2[12020] = {X 295.8472, Y 45.9528, Z -3.0000, A 0.000, B 0.000, C 0.000 }
gfCNCPoint2[12021] = {X 295.7293, Y 46.4221, Z -3.0000, A 0.000, B 0.000, C 0.000 }
gfCNCPoint2[12022] = {X 295.4314, Y 47.1714, Z -3.0000, A 0.000, B 0.000, C 0.000 }
gfCNCPoint2[12023] = {X 295.0142, Y 47.8614, Z -3.0000, A 0.000, B 0.000, C 0.000 }
gfCNCPoint2[12024] = {X 294.4890, Y 48.4733, Z -3.0000, A 0.000, B 0.000, C 0.000 }
gfCNCPoint2[12025] = {X 295.3745, Y 48.6761, Z -3.0000, A 0.000, B 0.000, C 0.000 }
gfCNCPoint2[12026] = {X 296.2371, Y 48.9610, Z -3.0000, A 0.000, B 0.000, C 0.000 }
gfCNCPoint2[12027] = {X 295.3782, Y 51.2021, Z -3.0000, A 0.000, B 0.000, C 0.000 }
gfCNCPoint2[12028] = {X 296.3502, Y 51.6595, Z -3.0000, A 0.000, B 0.000, C 0.000 }
gfCNCPoint2[12029] = {X 297.2443, Y 52.2549, Z -3.0000, A 0.000, B 0.000, C 0.000 }
gfCNCPoint2[12030] = {X 298.0411, Y 52.9754, Z -3.0000, A 0.000, B 0.000, C 0.000 }
gfCNCPoint2[12031] = {X 298.7231, Y 53.8053, Z -3.0000, A 0.000, B 0.000, C 0.000 }
gfCNCPoint2[12032] = {X 299.2946, Y 54.7645, Z -3.0000, A 0.000, B 0.000, C 0.000 }
gfCNCPoint2[12033] = {X 299.7126, Y 55.7997, Z -3.0000, A 0.000, B 0.000, C 0.000 }
gfCNCPoint2[12034] = {X 299.9675, Y 56.8868, Z -3.0000, A 0.000, B 0.000, C 0.000 }
gfCNCPoint2[12035] = {X 300.0531, Y 58.0000, Z -3.0000, A 0.000, B 0.000, C 0.000 }
gfCNCPoint2[12036] = {X 300.0531, Y 58.9451, Z -3.0000, A 0.000, B 0.000, C 0.000 }
gfCNCPoint2[12037] = {X 299.9645, Y 60.0545, Z -3.0000, A 0.000, B 0.000, C 0.000 }
gfCNCPoint2[12038] = {X 299.7082, Y 61.1375, Z -3.0000, A 0.000, B 0.000, C 0.000 }
gfCNCPoint2[12039] = {X 299.2902, Y 62.1689, Z -3.0000, A 0.000, B 0.000, C 0.000 }
gfCNCPoint2[12040] = {X 298.7202, Y 63.1248, Z -3.0000, A 0.000, B 0.000, C 0.000 }
gfCNCPoint2[12041] = {X 300.6818, Y 64.5076, Z -3.0000, A 0.000, B 0.000, C 0.000 }
gfCNCPoint2[12042] = {X 299.7821, Y 65.6039, Z -3.0000, A 0.000, B 0.000, C 0.000 }
gfCNCPoint2[12043] = {X 298.7321, Y 66.5573, Z -3.0000, A 0.000, B 0.000, C 0.000 }
gfCNCPoint2[12044] = {X 298.7321, Y 89.4423, Z -3.0000, A 0.000, B 0.000, C 0.000 }
gfCNCPoint2[12045] = {X 299.8288, Y 90.4466, Z -3.0000, A 0.000, B 0.000, C 0.000 }
gfCNCPoint2[12046] = {X 300.7594, Y 91.6065, Z -3.0000, A 0.000, B 0.000, C 0.000 }
gfCNCPoint2[12047] = {X 301.5020, Y 92.8950, Z -3.0000, A 0.000, B 0.000, C 0.000 }
gfCNCPoint2[12048] = {X 304.0676, Y 92.8950, Z -3.0000, A 0.000, B 0.000, C 0.000 }
gfCNCPoint2[12049] = {X 303.7100, Y 91.8995, Z -3.0000, A 0.000, B 0.000, C 0.000 }
gfCNCPoint2[12050] = {X 303.4139, Y 90.8840, Z -3.0000, A 0.000, B 0.000, C 0.000 }
gfCNCPoint2[12051] = {X 302.9749, Y 88.8129, Z -3.0000, A 0.000, B 0.000, C 0.000 }
gfCNCPoint2[12052] = {X 302.7149, Y 86.7118, Z -3.0000, A 0.000, B 0.000, C 0.000 }
gfCNCPoint2[12053] = {X 302.6361, Y 84.5962, Z -3.0000, A 0.000, B 0.000, C 0.000 }
gfCNCPoint2[12054] = {X 302.6373, Y 83.2276, Z -3.0000, A 0.000, B 0.000, C 0.000 }
gfCNCPoint2[12055] = {X 302.6373, Y 66.5625, Z -3.0000, A 0.000, B 0.000, C 0.000 }
gfCNCPoint2[12056] = {X 301.5839, Y 65.6071, Z -3.0000, A 0.000, B 0.000, C 0.000 }
